LIN {X 103.987,Y -19.308,Z -79.149,A -90.000,B 90.000,C 0.000} C_DIS
LIN {X 103.058,Y -19.308,Z -80.726,A -90.000,B 90.000,C 0.000} C_DIS
LIN {X 102.198,Y -19.308,Z -82.078,A -90.000,B 90.000,C 0.000} C_DIS
LIN {X 99.737,Y -19.308,Z -85.762,A -90.000,B 90.000,C 0.000} C_DIS
LIN {X 99.864,Y -19.308,Z -87.386,A -90.000,B 90.000,C 0.000} C_DIS
LIN {X 100.040,Y -19.308,Z -89.899,A -90.000,B 90.000,C 0.000} C_DIS
LIN {X 100.045,Y -19.308,Z -89.957,A -90.000,B 90.000,C 0.000} C_DIS
LIN {X 100.412,Y -19.308,Z -91.345,A -90.000,B 90.000,C 0.000} C_DIS
LIN {X 100.428,Y -19.308,Z -91.411,A -90.000,B 90.000,C 0.000} C_DIS
LIN {X 100.504,Y -19.308,Z -91.700,A -90.000,B 90.000,C 0.000} C_DIS
LIN {X 100.648,Y -19.308,Z -92.531,A -90.000,B 90.000,C 0.000} C_DIS
LIN {X 100.763,Y -19.308,Z -93.019,A -90.000,B 90.000,C 0.000} C_DIS
LIN {X 100.838,Y -19.308,Z -93.500,A -90.000,B 90.000,C 0.000} C_DIS
LIN {X 100.877,Y -19.308,Z -93.994,A -90.000,B 90.000,C 0.000} C_DIS
LIN {X 100.998,Y -19.308,Z -94.813,A -90.000,B 90.000,C 0.000} C_DIS
LIN {X 101.014,Y -19.308,Z -95.123,A -90.000,B 90.000,C 0.000} C_DIS
LIN {X 101.095,Y -19.308,Z -96.027,A -90.000,B 90.000,C 0.000} C_DIS
LIN {X 101.110,Y -19.308,Z -96.320,A -90.000,B 90.000,C 0.000} C_DIS
LIN {X 101.175,Y -19.308,Z -97.267,A -90.000,B 90.000,C 0.000} C_DIS
LIN {X 101.202,Y -19.308,Z -97.483,A -90.000,B 90.000,C 0.000} C_DIS
LIN {X 101.290,Y -19.308,Z -98.618,A -90.000,B 90.000,C 0.000} C_DIS
LIN {X 101.319,Y -19.308,Z -98.809,A -90.000,B 90.000,C 0.000} C_DIS
LIN {X 101.430,Y -19.308,Z -100.112,A -90.000,B 90.000,C 0.000} C_DIS
LIN {X 101.445,Y -19.308,Z -100.208,A -90.000,B 90.000,C 0.000} C_DIS
LIN {X 101.588,Y -19.308,Z -101.701,A -90.000,B 90.000,C 0.000} C_DIS
LIN {X 101.643,Y -19.308,Z -102.068,A -90.000,B 90.000,C 0.000} C_DIS
LIN {X 101.782,Y -19.308,Z -103.351,A -90.000,B 90.000,C 0.000} C_DIS
LIN {X 101.920,Y -19.308,Z -104.378,A -90.000,B 90.000,C 0.000} C_DIS
LIN {X 102.259,Y -19.308,Z -106.543,A -90.000,B 90.000,C 0.000} C_DIS
LIN {X 102.427,Y -19.308,Z -107.635,A -90.000,B 90.000,C 0.000} C_DIS
LIN {X 102.586,Y -19.308,Z -108.751,A -90.000,B 90.000,C 0.000} C_DIS
LIN {X 102.776,Y -19.308,Z -110.166,A -90.000,B 90.000,C 0.000} C_DIS
LIN {X 103.011,Y -19.308,Z -111.971,A -90.000,B 90.000,C 0.000} C_DIS
LIN {X 103.313,Y -19.308,Z -114.380,A -90.000,B 90.000,C 0.000} C_DIS
LIN {X 103.602,Y -19.308,Z -116.737,A -90.000,B 90.000,C 0.000} C_DIS
LIN {X 103.814,Y -19.308,Z -118.582,A -90.000,B 90.000,C 0.000} C_DIS
LIN {X 103.886,Y -19.308,Z -119.181,A -90.000,B 90.000,C 0.000} C_DIS
LIN {X 104.063,Y -19.308,Z -120.883,A -90.000,B 90.000,C 0.000} C_DIS
LIN {X 104.148,Y -19.308,Z -121.663,A -90.000,B 90.000,C 0.000} C_DIS
LIN {X 104.284,Y -19.308,Z -123.195,A -90.000,B 90.000,C 0.000} C_DIS
LIN {X 104.370,Y -19.308,Z -124.134,A -90.000,B 90.000,C 0.000} C_DIS
LIN {X 104.532,Y -19.308,Z -126.543,A -90.000,B 90.000,C 0.000} C_DIS
LIN {X 104.557,Y -19.308,Z -127.010,A -90.000,B 90.000,C 0.000} C_DIS
LIN {X 104.601,Y -19.308,Z -128.190,A -90.000,B 90.000,C 0.000} C_DIS
LIN {X 104.655,Y -19.308,Z -129.468,A -90.000,B 90.000,C 0.000} C_DIS
LIN {X 104.668,Y -19.308,Z -130.834,A -90.000,B 90.000,C 0.000} C_DIS
LIN {X 104.688,Y -19.308,Z -132.086,A -90.000,B 90.000,C 0.000} C_DIS
LIN {X 104.665,Y -19.308,Z -133.696,A -90.000,B 90.000,C 0.000} C_DIS
LIN {X 104.655,Y -19.308,Z -134.974,A -90.000,B 90.000,C 0.000} C_DIS
LIN {X 104.619,Y -19.308,Z -136.319,A -90.000,B 90.000,C 0.000} C_DIS
LIN {X 104.547,Y -19.308,Z -138.447,A -90.000,B 90.000,C 0.000} C_DIS
LIN {X 104.485,Y -19.308,Z -139.937,A -90.000,B 90.000,C 0.000} C_DIS
LIN {X 104.383,Y -19.308,Z -142.127,A -90.000,B 90.000,C 0.000} C_DIS
LIN {X 104.310,Y -19.308,Z -143.499,A -90.000,B 90.000,C 0.000} C_DIS
LIN {X 104.174,Y -19.308,Z -145.853,A -90.000,B 90.000,C 0.000} C_DIS
LIN {X 104.083,Y -19.308,Z -147.291,A -90.000,B 90.000,C 0.000} C_DIS
LIN {X 103.924,Y -19.308,Z -149.658,A -90.000,B 90.000,C 0.000} C_DIS
LIN {X 103.809,Y -19.308,Z -151.181,A -90.000,B 90.000,C 0.000} C_DIS
LIN {X 103.665,Y -19.308,Z -153.152,A -90.000,B 90.000,C 0.000} C_DIS
LIN {X 103.314,Y -19.308,Z -157.499,A -90.000,B 90.000,C 0.000} C_DIS
LIN {X 102.978,Y -19.308,Z -161.384,A -90.000,B 90.000,C 0.000} C_DIS
LIN {X 102.664,Y -19.308,Z -164.871,A -90.000,B 90.000,C 0.000} C_DIS
LIN {X 102.336,Y -19.308,Z -168.404,A -90.000,B 90.000,C 0.000} C_DIS
LIN {X 102.004,Y -19.308,Z -171.823,A -90.000,B 90.000,C 0.000} C_DIS
LIN {X 101.666,Y -19.308,Z -175.075,A -90.000,B 90.000,C 0.000} C_DIS
LIN {X 101.590,Y -19.308,Z -175.741,A -90.000,B 90.000,C 0.000} C_DIS
LIN {X 101.303,Y -19.308,Z -178.170,A -90.000,B 90.000,C 0.000} C_DIS
LIN {X 100.894,Y -19.308,Z -181.246,A -90.000,B 90.000,C 0.000} C_DIS
LIN {X 100.474,Y -19.308,Z -184.127,A -90.000,B 90.000,C 0.000} C_DIS
LIN {X 100.075,Y -19.308,Z -186.713,A -90.000,B 90.000,C 0.000} C_DIS
LIN {X 99.715,Y -19.308,Z -189.013,A -90.000,B 90.000,C 0.000} C_DIS
LIN {X 99.354,Y -19.308,Z -191.397,A -90.000,B 90.000,C 0.000} C_DIS
LIN {X 99.271,Y -19.308,Z -191.933,A -90.000,B 90.000,C 0.000} C_DIS
LIN {X 98.939,Y -19.308,Z -193.967,A -90.000,B 90.000,C 0.000} C_DIS
LIN {X 98.678,Y -19.308,Z -195.458,A -90.000,B 90.000,C 0.000} C_DIS
LIN {X 98.423,Y -19.308,Z -196.834,A -90.000,B 90.000,C 0.000} C_DIS
LIN {X 98.011,Y -19.308,Z -198.956,A -90.000,B 90.000,C 0.000} C_DIS
LIN {X 97.713,Y -19.308,Z -200.366,A -90.000,B 90.000,C 0.000} C_DIS
LIN {X 97.101,Y -19.308,Z -203.218,A -90.000,B 90.000,C 0.000} C_DIS
LIN {X 96.760,Y -19.308,Z -204.668,A -90.000,B 90.000,C 0.000} C_DIS
LIN {X 95.957,Y -19.308,Z -208.195,A -90.000,B 90.000,C 0.000} C_DIS
LIN {X 95.642,Y -19.308,Z -209.516,A -90.000,B 90.000,C 0.000} C_DIS
LIN {X 95.578,Y -19.308,Z -209.775,A -90.000,B 90.000,C 0.000} C_DIS
LIN {X 94.321,Y -19.308,Z -215.060,A -90.000,B 90.000,C 0.000} C_DIS
LIN {X 92.959,Y -19.308,Z -220.548,A -90.000,B 90.000,C 0.000} C_DIS
LIN {X 91.672,Y -19.308,Z -225.536,A -90.000,B 90.000,C 0.000} C_DIS
LIN {X 91.541,Y -19.308,Z -226.056,A -90.000,B 90.000,C 0.000} C_DIS
LIN {X 89.987,Y -19.308,Z -231.676,A -90.000,B 90.000,C 0.000} C_DIS
LIN {X 88.154,Y -19.308,Z -237.735,A -90.000,B 90.000,C 0.000} C_DIS
LIN {X 88.090,Y -19.308,Z -237.937,A -90.000,B 90.000,C 0.000} C_DIS
LIN {X 86.454,Y -19.308,Z -242.832,A -90.000,B 90.000,C 0.000} C_DIS
LIN {X 86.214,Y -19.308,Z -243.561,A -90.000,B 90.000,C 0.000} C_DIS
LIN {X 86.214,Y -60.000,Z -243.561,A -90.000,B 90.000,C 0.000} C_DIS
LIN {X 100.091,Y -60.000,Z -90.101,A -90.000,B 90.000,C 0.000} C_DIS
LIN {X 100.091,Y -17.308,Z -90.101,A -90.000,B 90.000,C 0.000} C_DIS
LIN {X 100.230,Y -17.309,Z -90.520,A -90.000,B 90.000,C 0.000} C_DIS
LIN {X 100.336,Y -17.309,Z -90.804,A -90.000,B 90.000,C 0.000} C_DIS
LIN {X 100.668,Y -17.314,Z -91.753,A -90.000,B 90.000,C 0.000} C_DIS
LIN {X 100.794,Y -17.318,Z -92.235,A -90.000,B 90.000,C 0.000} C_DIS
LIN {X 100.884,Y -17.319,Z -92.622,A -90.000,B 90.000,C 0.000} C_DIS
LIN {X 100.988,Y -17.321,Z -92.984,A -90.000,B 90.000,C 0.000} C_DIS
LIN {X 101.100,Y -17.327,Z -93.411,A -90.000,B 90.000,C 0.000} C_DIS
LIN {X 101.168,Y -17.331,Z -93.853,A -90.000,B 90.000,C 0.000} C_DIS
LIN {X 101.322,Y -17.339,Z -94.610,A -90.000,B 90.000,C 0.000} C_DIS
LIN {X 101.351,Y -17.340,Z -94.795,A -90.000,B 90.000,C 0.000} C_DIS
LIN {X 101.396,Y -17.345,Z -95.095,A -90.000,B 90.000,C 0.000} C_DIS
LIN {X 101.414,Y -17.345,Z -95.293,A -90.000,B 90.000,C 0.000} C_DIS
LIN {X 101.528,Y -17.355,Z -96.069,A -90.000,B 90.000,C 0.000} C_DIS
LIN {X 101.546,Y -17.358,Z -96.196,A -90.000,B 90.000,C 0.000} C_DIS
LIN {X 101.560,Y -17.358,Z -96.404,A -90.000,B 90.000,C 0.000} C_DIS
LIN {X 101.676,Y -17.369,Z -97.317,A -90.000,B 90.000,C 0.000} C_DIS
LIN {X 101.756,Y -17.377,Z -97.898,A -90.000,B 90.000,C 0.000} C_DIS
LIN {X 101.825,Y -17.386,Z -98.396,A -90.000,B 90.000,C 0.000} C_DIS
LIN {X 101.854,Y -17.387,Z -98.629,A -90.000,B 90.000,C 0.000} C_DIS
LIN {X 101.860,Y -17.387,Z -98.688,A -90.000,B 90.000,C 0.000} C_DIS
LIN {X 101.918,Y -17.392,Z -99.080,A -90.000,B 90.000,C 0.000} C_DIS
LIN {X 102.046,Y -17.409,Z -99.960,A -90.000,B 90.000,C 0.000} C_DIS
LIN {X 102.058,Y -17.408,Z -100.094,A -90.000,B 90.000,C 0.000} C_DIS
LIN {X 102.260,Y -17.433,Z -101.436,A -90.000,B 90.000,C 0.000} C_DIS
LIN {X 102.287,Y -17.431,Z -101.711,A -90.000,B 90.000,C 0.000} C_DIS
LIN {X 102.331,Y -17.432,Z -101.994,A -90.000,B 90.000,C 0.000} C_DIS
LIN {X 102.532,Y -17.453,Z -103.332,A -90.000,B 90.000,C 0.000} C_DIS
LIN {X 102.578,Y -17.454,Z -103.640,A -90.000,B 90.000,C 0.000} C_DIS
LIN {X 102.603,Y -17.453,Z -103.849,A -90.000,B 90.000,C 0.000} C_DIS
LIN {X 102.667,Y -17.457,Z -104.269,A -90.000,B 90.000,C 0.000} C_DIS
LIN {X 102.901,Y -17.457,Z -105.750,A -90.000,B 90.000,C 0.000} C_DIS
LIN {X 103.122,Y -17.455,Z -107.208,A -90.000,B 90.000,C 0.000} C_DIS
LIN {X 103.352,Y -17.458,Z -108.760,A -90.000,B 90.000,C 0.000} C_DIS
LIN {X 103.439,Y -17.459,Z -109.387,A -90.000,B 90.000,C 0.000} C_DIS
LIN {X 103.665,Y -17.461,Z -111.052,A -90.000,B 90.000,C 0.000} C_DIS
LIN {X 103.740,Y -17.462,Z -111.617,A -90.000,B 90.000,C 0.000} C_DIS
LIN {X 104.045,Y -17.461,Z -114.051,A -90.000,B 90.000,C 0.000} C_DIS
LIN {X 104.152,Y -17.457,Z -115.015,A -90.000,B 90.000,C 0.000} C_DIS
LIN {X 104.226,Y -17.455,Z -115.644,A -90.000,B 90.000,C 0.000} C_DIS
LIN {X 104.332,Y -17.453,Z -116.545,A -90.000,B 90.000,C 0.000} C_DIS
LIN {X 104.387,Y -17.450,Z -117.097,A -90.000,B 90.000,C 0.000} C_DIS
LIN {X 104.604,Y -17.443,Z -119.102,A -90.000,B 90.000,C 0.000} C_DIS
LIN {X 104.811,Y -17.437,Z -121.240,A -90.000,B 90.000,C 0.000} C_DIS
LIN {X 104.850,Y -17.436,Z -121.606,A -90.000,B 90.000,C 0.000} C_DIS
LIN {X 105.001,Y -17.432,Z -123.421,A -90.000,B 90.000,C 0.000} C_DIS
LIN {X 105.063,Y -17.432,Z -124.100,A -90.000,B 90.000,C 0.000} C_DIS
LIN {X 105.228,Y -17.433,Z -126.534,A -90.000,B 90.000,C 0.000} C_DIS
LIN {X 105.256,Y -17.433,Z -127.072,A -90.000,B 90.000,C 0.000} C_DIS
LIN {X 105.363,Y -17.438,Z -129.492,A -90.000,B 90.000,C 0.000} C_DIS
LIN {X 105.387,Y -17.442,Z -130.825,A -90.000,B 90.000,C 0.000} C_DIS
LIN {X 105.414,Y -17.445,Z -132.132,A -90.000,B 90.000,C 0.000} C_DIS
LIN {X 105.404,Y -17.450,Z -133.704,A -90.000,B 90.000,C 0.000} C_DIS
LIN {X 105.400,Y -17.453,Z -135.091,A -90.000,B 90.000,C 0.000} C_DIS
LIN {X 105.360,Y -17.458,Z -136.853,A -90.000,B 90.000,C 0.000} C_DIS
LIN {X 105.316,Y -17.462,Z -138.473,A -90.000,B 90.000,C 0.000} C_DIS
LIN {X 105.222,Y -17.468,Z -140.956,A -90.000,B 90.000,C 0.000} C_DIS
LIN {X 105.169,Y -17.472,Z -142.260,A -90.000,B 90.000,C 0.000} C_DIS
LIN {X 105.092,Y -17.474,Z -143.764,A -90.000,B 90.000,C 0.000} C_DIS
LIN {X 104.980,Y -17.478,Z -145.900,A -90.000,B 90.000,C 0.000} C_DIS
LIN {X 104.775,Y -17.481,Z -149.127,A -90.000,B 90.000,C 0.000} C_DIS
LIN {X 104.729,Y -17.482,Z -149.845,A -90.000,B 90.000,C 0.000} C_DIS
LIN {X 104.440,Y -17.481,Z -153.671,A -90.000,B 90.000,C 0.000} C_DIS
LIN {X 104.110,Y -17.475,Z -157.564,A -90.000,B 90.000,C 0.000} C_DIS
LIN {X 103.752,Y -17.466,Z -161.459,A -90.000,B 90.000,C 0.000} C_DIS
LIN {X 103.351,Y -17.454,Z -165.582,A -90.000,B 90.000,C 0.000} C_DIS
LIN {X 102.981,Y -17.446,Z -169.296,A -90.000,B 90.000,C 0.000} C_DIS
LIN {X 102.710,Y -17.440,Z -171.918,A -90.000,B 90.000,C 0.000} C_DIS
LIN {X 102.535,Y -17.436,Z -173.522,A -90.000,B 90.000,C 0.000} C_DIS
LIN {X 102.352,Y -17.432,Z -175.180,A -90.000,B 90.000,C 0.000} C_DIS
LIN {X 101.981,Y -17.429,Z -178.250,A -90.000,B 90.000,C 0.000} C_DIS
LIN {X 101.603,Y -17.426,Z -181.040,A -90.000,B 90.000,C 0.000} C_DIS
LIN {X 101.539,Y -17.425,Z -181.488,A -90.000,B 90.000,C 0.000} C_DIS
LIN {X 101.155,Y -17.423,Z -184.085,A -90.000,B 90.000,C 0.000} C_DIS
LIN {X 100.474,Y -17.418,Z -188.393,A -90.000,B 90.000,C 0.000} C_DIS
LIN {X 100.361,Y -17.418,Z -189.114,A -90.000,B 90.000,C 0.000} C_DIS
LIN {X 99.996,Y -17.417,Z -191.494,A -90.000,B 90.000,C 0.000} C_DIS
LIN {X 99.965,Y -17.416,Z -191.688,A -90.000,B 90.000,C 0.000} C_DIS
LIN {X 99.583,Y -17.418,Z -194.072,A -90.000,B 90.000,C 0.000} C_DIS
LIN {X 99.476,Y -17.419,Z -194.709,A -90.000,B 90.000,C 0.000} C_DIS
LIN {X 99.324,Y -17.419,Z -195.572,A -90.000,B 90.000,C 0.000} C_DIS
LIN {X 99.078,Y -17.423,Z -196.955,A -90.000,B 90.000,C 0.000} C_DIS
LIN {X 98.888,Y -17.427,Z -198.002,A -90.000,B 90.000,C 0.000} C_DIS
LIN {X 98.676,Y -17.427,Z -199.085,A -90.000,B 90.000,C 0.000} C_DIS
LIN {X 98.394,Y -17.433,Z -200.509,A -90.000,B 90.000,C 0.000} C_DIS
LIN {X 98.106,Y -17.443,Z -201.970,A -90.000,B 90.000,C 0.000} C_DIS
LIN {X 97.805,Y -17.442,Z -203.369,A -90.000,B 90.000,C 0.000} C_DIS
LIN {X 97.484,Y -17.452,Z -204.839,A -90.000,B 90.000,C 0.000} C_DIS
LIN {X 97.050,Y -17.466,Z -206.904,A -90.000,B 90.000,C 0.000} C_DIS
LIN {X 96.867,Y -17.471,Z -207.754,A -90.000,B 90.000,C 0.000} C_DIS
LIN {X 96.726,Y -17.470,Z -208.370,A -90.000,B 90.000,C 0.000} C_DIS
LIN {X 96.421,Y -17.475,Z -209.701,A -90.000,B 90.000,C 0.000} C_DIS
LIN {X 95.655,Y -17.498,Z -213.123,A -90.000,B 90.000,C 0.000} C_DIS
LIN {X 95.147,Y -17.498,Z -215.256,A -90.000,B 90.000,C 0.000} C_DIS
LIN {X 94.309,Y -17.515,Z -218.783,A -90.000,B 90.000,C 0.000} C_DIS
LIN {X 93.950,Y -17.518,Z -220.254,A -90.000,B 90.000,C 0.000} C_DIS
LIN {X 93.823,Y -17.517,Z -220.763,A -90.000,B 90.000,C 0.000} C_DIS
LIN {X 93.724,Y -17.517,Z -221.147,A -90.000,B 90.000,C 0.000} C_DIS
LIN {X 92.458,Y -17.526,Z -226.130,A -90.000,B 90.000,C 0.000} C_DIS
LIN {X 92.352,Y -17.525,Z -226.517,A -90.000,B 90.000,C 0.000} C_DIS
LIN {X 90.897,Y -17.526,Z -231.788,A -90.000,B 90.000,C 0.000} C_DIS
LIN {X 90.724,Y -17.524,Z -232.363,A -90.000,B 90.000,C 0.000} C_DIS
LIN {X 89.062,Y -17.525,Z -237.861,A -90.000,B 90.000,C 0.000} C_DIS
LIN {X 88.983,Y -17.524,Z -238.109,A -90.000,B 90.000,C 0.000} C_DIS
LIN {X 87.179,Y -17.531,Z -243.561,A -90.000,B 90.000,C 0.000} C_DIS
LIN {X 87.179,Y -60.000,Z -243.561,A -90.000,B 90.000,C 0.000} C_DIS
LIN {X -110.313,Y -60.000,Z -243.561,A -90.000,B 90.000,C 0.000} C_DIS
LIN {X -110.313,Y -18.479,Z -243.561,A -90.000,B 90.000,C 0.000} C_DIS
LIN {X -110.301,Y -18.455,Z -243.517,A -90.000,B 90.000,C 0.000} C_DIS
LIN {X -110.261,Y -18.391,Z -243.388,A -90.000,B 90.000,C 0.000} C_DIS
LIN {X -110.203,Y -18.323,Z -243.242,A -90.000,B 90.000,C 0.000} C_DIS
LIN {X -110.174,Y -18.295,Z -243.177,A -90.000,B 90.000,C 0.000} C_DIS
LIN {X -109.840,Y -18.124,Z -242.677,A -90.000,B 90.000,C 0.000} C_DIS
LIN {X -109.452,Y -18.069,Z -242.319,A -90.000,B 90.000,C 0.000} C_DIS
LIN {X -109.374,Y -18.068,Z -242.263,A -90.000,B 90.000,C 0.000} C_DIS
LIN {X -108.603,Y -18.076,Z -241.732,A -90.000,B 90.000,C 0.000} C_DIS
LIN {X -106.834,Y -18.082,Z -240.498,A -90.000,B 90.000,C 0.000} C_DIS
LIN {X -100.205,Y -18.099,Z -235.847,A -90.000,B 90.000,C 0.000} C_DIS
LIN {X -97.781,Y -18.102,Z -234.146,A -90.000,B 90.000,C 0.000} C_DIS
LIN {X -93.938,Y -18.110,Z -231.476,A -90.000,B 90.000,C 0.000} C_DIS
LIN {X -89.899,Y -18.111,Z -228.673,A -90.000,B 90.000,C 0.000} C_DIS
LIN {X -89.665,Y -18.110,Z -228.511,A -90.000,B 90.000,C 0.000} C_DIS
LIN {X -87.245,Y -18.114,Z -226.866,A -90.000,B 90.000,C 0.000} C_DIS
LIN {X -81.874,Y -18.116,Z -223.210,A -90.000,B 90.000,C 0.000} C_DIS
LIN {X -81.580,Y -18.114,Z -223.011,A -90.000,B 90.000,C 0.000} C_DIS
LIN {X -76.713,Y -18.118,Z -219.783,A -90.000,B 90.000,C 0.000} C_DIS
LIN {X -73.418,Y -18.109,Z -217.608,A -90.000,B 90.000,C 0.000} C_DIS
LIN {X -70.830,Y -18.099,Z -215.910,A -90.000,B 90.000,C 0.000} C_DIS
LIN {X -65.406,Y -18.087,Z -212.367,A -90.000,B 90.000,C 0.000} C_DIS
LIN {X -60.511,Y -18.066,Z -209.130,A -90.000,B 90.000,C 0.000} C_DIS
LIN {X -58.236,Y -18.060,Z -207.634,A -90.000,B 90.000,C 0.000} C_DIS
LIN {X -57.950,Y -18.062,Z -207.444,A -90.000,B 90.000,C 0.000} C_DIS
LIN {X -51.703,Y -18.026,Z -203.201,A -90.000,B 90.000,C 0.000} C_DIS
LIN {X -51.585,Y -18.027,Z -203.119,A -90.000,B 90.000,C 0.000} C_DIS
LIN {X -46.435,Y -18.015,Z -199.479,A -90.000,B 90.000,C 0.000} C_DIS
LIN {X -46.154,Y -18.018,Z -199.276,A -90.000,B 90.000,C 0.000} C_DIS
LIN {X -43.931,Y -18.008,Z -197.626,A -90.000,B 90.000,C 0.000} C_DIS
LIN {X -41.923,Y -17.985,Z -196.152,A -90.000,B 90.000,C 0.000} C_DIS
LIN {X -41.724,Y -17.985,Z -196.003,A -90.000,B 90.000,C 0.000} C_DIS
LIN {X -40.829,Y -17.980,Z -195.324,A -90.000,B 90.000,C 0.000} C_DIS
LIN {X -38.690,Y -17.954,Z -193.683,A -90.000,B 90.000,C 0.000} C_DIS
LIN {X -38.089,Y -17.943,Z -193.227,A -90.000,B 90.000,C 0.000} C_DIS
LIN {X -36.620,Y -17.931,Z -192.090,A -90.000,B 90.000,C 0.000} C_DIS
LIN {X -34.749,Y -17.901,Z -190.626,A -90.000,B 90.000,C 0.000} C_DIS
LIN {X -32.943,Y -17.881,Z -189.202,A -90.000,B 90.000,C 0.000} C_DIS
LIN {X -31.630,Y -17.878,Z -188.178,A -90.000,B 90.000,C 0.000} C_DIS
LIN {X -31.435,Y -17.879,Z -188.023,A -90.000,B 90.000,C 0.000} C_DIS
LIN {X -30.006,Y -17.868,Z -186.865,A -90.000,B 90.000,C 0.000} C_DIS
LIN {X -28.713,Y -17.868,Z -185.829,A -90.000,B 90.000,C 0.000} C_DIS
LIN {X -28.525,Y -17.871,Z -185.673,A -90.000,B 90.000,C 0.000} C_DIS
LIN {X -27.122,Y -17.861,Z -184.479,A -90.000,B 90.000,C 0.000} C_DIS
LIN {X -25.979,Y -17.862,Z -183.517,A -90.000,B 90.000,C 0.000} C_DIS
LIN {X -24.802,Y -17.852,Z -182.443,A -90.000,B 90.000,C 0.000} C_DIS
LIN {X -23.613,Y -17.853,Z -181.372,A -90.000,B 90.000,C 0.000} C_DIS
LIN {X -23.524,Y -17.855,Z -181.286,A -90.000,B 90.000,C 0.000} C_DIS
LIN {X -22.591,Y -17.854,Z -180.371,A -90.000,B 90.000,C 0.000} C_DIS
LIN {X -21.251,Y -17.839,Z -179.039,A -90.000,B 90.000,C 0.000} C_DIS
LIN {X -21.040,Y -17.844,Z -178.818,A -90.000,B 90.000,C 0.000} C_DIS
LIN {X -20.425,Y -17.843,Z -178.154,A -90.000,B 90.000,C 0.000} C_DIS
LIN {X -19.010,Y -17.825,Z -176.606,A -90.000,B 90.000,C 0.000} C_DIS
LIN {X -18.887,Y -17.828,Z -176.463,A -90.000,B 90.000,C 0.000} C_DIS
LIN {X -18.374,Y -17.828,Z -175.846,A -90.000,B 90.000,C 0.000} C_DIS
LIN {X -17.081,Y -17.809,Z -174.270,A -90.000,B 90.000,C 0.000} C_DIS
LIN {X -16.818,Y -17.817,Z -173.925,A -90.000,B 90.000,C 0.000} C_DIS
LIN {X -16.274,Y -17.819,Z -173.186,A -90.000,B 90.000,C 0.000} C_DIS
LIN {X -15.242,Y -17.798,Z -171.754,A -90.000,B 90.000,C 0.000} C_DIS
LIN {X -15.058,Y -17.806,Z -171.475,A -90.000,B 90.000,C 0.000} C_DIS
LIN {X -14.670,Y -17.808,Z -170.864,A -90.000,B 90.000,C 0.000} C_DIS
LIN {X -13.644,Y -17.777,Z -169.200,A -90.000,B 90.000,C 0.000} C_DIS
LIN {X -13.389,Y -17.791,Z -168.737,A -90.000,B 90.000,C 0.000} C_DIS
LIN {X -13.310,Y -17.791,Z -168.587,A -90.000,B 90.000,C 0.000} C_DIS
LIN {X -12.460,Y -17.750,Z -166.906,A -90.000,B 90.000,C 0.000} C_DIS
LIN {X -12.399,Y -17.751,Z -166.777,A -90.000,B 90.000,C 0.000} C_DIS
LIN {X -12.219,Y -17.765,Z -166.355,A -90.000,B 90.000,C 0.000} C_DIS
LIN {X -11.645,Y -17.726,Z -164.814,A -90.000,B 90.000,C 0.000} C_DIS
LIN {X -11.564,Y -17.727,Z -164.573,A -90.000,B 90.000,C 0.000} C_DIS
LIN {X -11.483,Y -17.743,Z -164.266,A -90.000,B 90.000,C 0.000} C_DIS
LIN {X -11.234,Y -17.711,Z -163.012,A -90.000,B 90.000,C 0.000} C_DIS
LIN {X -11.233,Y -17.735,Z -162.809,A -90.000,B 90.000,C 0.000} C_DIS
LIN {X -11.258,Y -17.724,Z -162.439,A -90.000,B 90.000,C 0.000} C_DIS
LIN {X -11.277,Y -17.714,Z -162.137,A -90.000,B 90.000,C 0.000} C_DIS
LIN {X -11.311,Y -17.679,Z -161.927,A -90.000,B 90.000,C 0.000} C_DIS
LIN {X -11.431,Y -17.667,Z -161.591,A -90.000,B 90.000,C 0.000} C_DIS
LIN {X -11.573,Y -17.618,Z -161.265,A -90.000,B 90.000,C 0.000} C_DIS
LIN {X -11.777,Y -17.616,Z -160.935,A -90.000,B 90.000,C 0.000} C_DIS
LIN {X -12.055,Y -17.570,Z -160.529,A -90.000,B 90.000,C 0.000} C_DIS
LIN {X -12.189,Y -17.564,Z -160.370,A -90.000,B 90.000,C 0.000} C_DIS
LIN {X -12.579,Y -17.562,Z -159.895,A -90.000,B 90.000,C 0.000} C_DIS
LIN {X -12.689,Y -17.558,Z -159.753,A -90.000,B 90.000,C 0.000} C_DIS
LIN {X -12.856,Y -17.547,Z -159.541,A -90.000,B 90.000,C 0.000} C_DIS
LIN {X -12.904,Y -17.543,Z -159.475,A -90.000,B 90.000,C 0.000} C_DIS
LIN {X -13.256,Y -17.539,Z -159.079,A -90.000,B 90.000,C 0.000} C_DIS
LIN {X -13.618,Y -17.525,Z -158.677,A -90.000,B 90.000,C 0.000} C_DIS
LIN {X -13.890,Y -17.505,Z -158.340,A -90.000,B 90.000,C 0.000} C_DIS
LIN {X -14.445,Y -17.501,Z -157.763,A -90.000,B 90.000,C 0.000} C_DIS
LIN {X -14.736,Y -17.492,Z -157.465,A -90.000,B 90.000,C 0.000} C_DIS
LIN {X -15.053,Y -17.472,Z -157.099,A -90.000,B 90.000,C 0.000} C_DIS
LIN {X -15.852,Y -17.469,Z -156.326,A -90.000,B 90.000,C 0.000} C_DIS
LIN {X -16.143,Y -17.462,Z -156.031,A -90.000,B 90.000,C 0.000} C_DIS
LIN {X -16.300,Y -17.456,Z -155.872,A -90.000,B 90.000,C 0.000} C_DIS
LIN {X -16.598,Y -17.443,Z -155.560,A -90.000,B 90.000,C 0.000} C_DIS
LIN {X -17.901,Y -17.442,Z -154.370,A -90.000,B 90.000,C 0.000} C_DIS
LIN {X -18.334,Y -17.434,Z -153.951,A -90.000,B 90.000,C 0.000} C_DIS
LIN {X -18.608,Y -17.426,Z -153.686,A -90.000,B 90.000,C 0.000} C_DIS
LIN {X -20.437,Y -17.425,Z -152.079,A -90.000,B 90.000,C 0.000} C_DIS
LIN {X -21.457,Y -17.414,Z -151.147,A -90.000,B 90.000,C 0.000} C_DIS
LIN {X -21.590,Y -17.412,Z -151.026,A -90.000,B 90.000,C 0.000} C_DIS
LIN {X -23.480,Y -17.412,Z -149.291,A -90.000,B 90.000,C 0.000} C_DIS
LIN {X -24.708,Y -17.403,Z -148.131,A -90.000,B 90.000,C 0.000} C_DIS
LIN {X -25.063,Y -17.402,Z -147.781,A -90.000,B 90.000,C 0.000} C_DIS
LIN {X -27.238,Y -17.403,Z -145.567,A -90.000,B 90.000,C 0.000} C_DIS
LIN {X -28.146,Y -17.398,Z -144.626,A -90.000,B 90.000,C 0.000} C_DIS
LIN {X -28.313,Y -17.396,Z -144.448,A -90.000,B 90.000,C 0.000} C_DIS
LIN {X -28.459,Y -17.396,Z -144.284,A -90.000,B 90.000,C 0.000} C_DIS
LIN {X -31.251,Y -17.401,Z -140.928,A -90.000,B 90.000,C 0.000} C_DIS
LIN {X -31.512,Y -17.400,Z -140.610,A -90.000,B 90.000,C 0.000} C_DIS
LIN {X -31.755,Y -17.395,Z -140.285,A -90.000,B 90.000,C 0.000} C_DIS
LIN {X -31.800,Y -17.396,Z -140.223,A -90.000,B 90.000,C 0.000} C_DIS
LIN {X -31.998,Y -17.394,Z -139.910,A -90.000,B 90.000,C 0.000} C_DIS
LIN {X -33.208,Y -17.397,Z -138.027,A -90.000,B 90.000,C 0.000} C_DIS
LIN {X -34.363,Y -17.399,Z -136.214,A -90.000,B 90.000,C 0.000} C_DIS
LIN {X -34.522,Y -17.396,Z -135.946,A -90.000,B 90.000,C 0.000} C_DIS
LIN {X -35.291,Y -17.395,Z -134.451,A -90.000,B 90.000,C 0.000} C_DIS
LIN {X -36.136,Y -17.394,Z -132.804,A -90.000,B 90.000,C 0.000} C_DIS
LIN {X -36.693,Y -17.395,Z -131.712,A -90.000,B 90.000,C 0.000} C_DIS
LIN {X -36.805,Y -17.392,Z -131.461,A -90.000,B 90.000,C 0.000} C_DIS
LIN {X -37.879,Y -17.391,Z -128.993,A -90.000,B 90.000,C 0.000} C_DIS
LIN {X -38.306,Y -17.391,Z -128.012,A -90.000,B 90.000,C 0.000} C_DIS
LIN {X -38.458,Y -17.388,Z -127.638,A -90.000,B 90.000,C 0.000} C_DIS
LIN {X -39.565,Y -17.381,Z -124.911,A -90.000,B 90.000,C 0.000} C_DIS
LIN {X -39.737,Y -17.380,Z -124.479,A -90.000,B 90.000,C 0.000} C_DIS
LIN {X -40.078,Y -17.375,Z -123.681,A -90.000,B 90.000,C 0.000} C_DIS
LIN {X -40.355,Y -17.368,Z -123.027,A -90.000,B 90.000,C 0.000} C_DIS
LIN {X -40.551,Y -17.362,Z -122.565,A -90.000,B 90.000,C 0.000} C_DIS
LIN {X -40.915,Y -17.357,Z -121.814,A -90.000,B 90.000,C 0.000} C_DIS
LIN {X -41.064,Y -17.353,Z -121.508,A -90.000,B 90.000,C 0.000} C_DIS
LIN {X -41.384,Y -17.349,Z -120.906,A -90.000,B 90.000,C 0.000} C_DIS
LIN {X -41.550,Y -17.349,Z -120.630,A -90.000,B 90.000,C 0.000} C_DIS
LIN {X -41.646,Y -17.347,Z -120.472,A -90.000,B 90.000,C 0.000} C_DIS
LIN {X -42.217,Y -17.344,Z -119.585,A -90.000,B 90.000,C 0.000} C_DIS
LIN {X -42.411,Y -17.347,Z -119.318,A -90.000,B 90.000,C 0.000} C_DIS
LIN {X -42.625,Y -17.346,Z -119.027,A -90.000,B 90.000,C 0.000} C_DIS
LIN {X -43.316,Y -17.345,Z -118.108,A -90.000,B 90.000,C 0.000} C_DIS
LIN {X -44.066,Y -17.351,Z -117.176,A -90.000,B 90.000,C 0.000} C_DIS
LIN {X -45.345,Y -17.355,Z -115.589,A -90.000,B 90.000,C 0.000} C_DIS
LIN {X -47.502,Y -17.366,Z -112.941,A -90.000,B 90.000,C 0.000} C_DIS
LIN {X -48.901,Y -17.369,Z -111.186,A -90.000,B 90.000,C 0.000} C_DIS
LIN {X -50.009,Y -17.374,Z -109.806,A -90.000,B 90.000,C 0.000} C_DIS
LIN {X -50.851,Y -17.373,Z -108.717,A -90.000,B 90.000,C 0.000} C_DIS
LIN {X -51.895,Y -17.377,Z -107.362,A -90.000,B 90.000,C 0.000} C_DIS
LIN {X -52.606,Y -17.378,Z -106.436,A -90.000,B 90.000,C 0.000} C_DIS
LIN {X -52.812,Y -17.377,Z -106.158,A -90.000,B 90.000,C 0.000} C_DIS
LIN {X -53.083,Y -17.374,Z -105.789,A -90.000,B 90.000,C 0.000} C_DIS
LIN {X -54.105,Y -17.373,Z -104.390,A -90.000,B 90.000,C 0.000} C_DIS
LIN {X -54.659,Y -17.370,Z -103.630,A -90.000,B 90.000,C 0.000} C_DIS
LIN {X -55.391,Y -17.368,Z -102.640,A -90.000,B 90.000,C 0.000} C_DIS
LIN {X -55.998,Y -17.365,Z -101.794,A -90.000,B 90.000,C 0.000} C_DIS
LIN {X -57.058,Y -17.364,Z -100.341,A -90.000,B 90.000,C 0.000} C_DIS
LIN {X -57.561,Y -17.361,Z -99.651,A -90.000,B 90.000,C 0.000} C_DIS
LIN {X -58.119,Y -17.359,Z -98.896,A -90.000,B 90.000,C 0.000} C_DIS
LIN {X -58.965,Y -17.355,Z -97.746,A -90.000,B 90.000,C 0.000} C_DIS
LIN {X -59.895,Y -17.355,Z -96.509,A -90.000,B 90.000,C 0.000} C_DIS
LIN {X -60.318,Y -17.356,Z -95.953,A -90.000,B 90.000,C 0.000} C_DIS
LIN {X -61.327,Y -17.356,Z -94.642,A -90.000,B 90.000,C 0.000} C_DIS
LIN {X -61.836,Y -17.354,Z -93.978,A -90.000,B 90.000,C 0.000} C_DIS
LIN {X -62.043,Y -17.354,Z -93.713,A -90.000,B 90.000,C 0.000} C_DIS
LIN {X -62.829,Y -17.355,Z -92.738,A -90.000,B 90.000,C 0.000} C_DIS
LIN {X -63.344,Y -17.355,Z -92.100,A -90.000,B 90.000,C 0.000} C_DIS
LIN {X -64.006,Y -17.356,Z -91.284,A -90.000,B 90.000,C 0.000} C_DIS
LIN {X -64.320,Y -17.360,Z -90.921,A -90.000,B 90.000,C 0.000} C_DIS
LIN {X -64.715,Y -17.361,Z -90.465,A -90.000,B 90.000,C 0.000} C_DIS
LIN {X -65.741,Y -17.363,Z -89.269,A -90.000,B 90.000,C 0.000} C_DIS
LIN {X -66.297,Y -17.367,Z -88.666,A -90.000,B 90.000,C 0.000} C_DIS
LIN {X -67.110,Y -17.370,Z -87.782,A -90.000,B 90.000,C 0.000} C_DIS
LIN {X -67.323,Y -17.370,Z -87.551,A -90.000,B 90.000,C 0.000} C_DIS
LIN {X -67.599,Y -17.377,Z -87.283,A -90.000,B 90.000,C 0.000} C_DIS
LIN {X -67.867,Y -17.381,Z -87.018,A -90.000,B 90.000,C 0.000} C_DIS
LIN {X -69.003,Y -17.389,Z -85.867,A -90.000,B 90.000,C 0.000} C_DIS
LIN {X -69.685,Y -17.404,Z -85.221,A -90.000,B 90.000,C 0.000} C_DIS
LIN {X -70.646,Y -17.422,Z -84.311,A -90.000,B 90.000,C 0.000} C_DIS
LIN {X -70.930,Y -17.431,Z -84.056,A -90.000,B 90.000,C 0.000} C_DIS
LIN {X -71.415,Y -17.448,Z -83.627,A -90.000,B 90.000,C 0.000} C_DIS
LIN {X -71.768,Y -17.458,Z -83.316,A -90.000,B 90.000,C 0.000} C_DIS
LIN {X -72.443,Y -17.476,Z -82.714,A -90.000,B 90.000,C 0.000} C_DIS
LIN {X -72.803,Y -17.495,Z -82.421,A -90.000,B 90.000,C 0.000} C_DIS
LIN {X -73.068,Y -17.506,Z -82.206,A -90.000,B 90.000,C 0.000} C_DIS
LIN {X -74.140,Y -17.542,Z -81.346,A -90.000,B 90.000,C 0.000} C_DIS
LIN {X -74.232,Y -17.546,Z -81.275,A -90.000,B 90.000,C 0.000} C_DIS
LIN {X -74.523,Y -17.569,Z -81.071,A -90.000,B 90.000,C 0.000} C_DIS
LIN {X -75.117,Y -17.586,Z -80.674,A -90.000,B 90.000,C 0.000} C_DIS
LIN {X -75.460,Y -17.598,Z -80.451,A -90.000,B 90.000,C 0.000} C_DIS
LIN {X -75.812,Y -17.575,Z -80.249,A -90.000,B 90.000,C 0.000} C_DIS
LIN {X -75.989,Y -17.574,Z -80.165,A -90.000,B 90.000,C 0.000} C_DIS
LIN {X -76.378,Y -17.572,Z -79.985,A -90.000,B 90.000,C 0.000} C_DIS
LIN {X -77.347,Y -17.510,Z -79.572,A -90.000,B 90.000,C 0.000} C_DIS
LIN {X -78.122,Y -17.474,Z -79.275,A -90.000,B 90.000,C 0.000} C_DIS
LIN {X -78.515,Y -17.461,Z -79.122,A -90.000,B 90.000,C 0.000} C_DIS
LIN {X -78.841,Y -17.448,Z -78.988,A -90.000,B 90.000,C 0.000} C_DIS
LIN {X -79.089,Y -17.444,Z -78.890,A -90.000,B 90.000,C 0.000} C_DIS
LIN {X -79.673,Y -17.437,Z -78.652,A -90.000,B 90.000,C 0.000} C_DIS
LIN {X -80.856,Y -17.410,Z -78.129,A -90.000,B 90.000,C 0.000} C_DIS
LIN {X -81.273,Y -17.404,Z -77.912,A -90.000,B 90.000,C 0.000} C_DIS
LIN {X -81.542,Y -17.402,Z -77.765,A -90.000,B 90.000,C 0.000} C_DIS
LIN {X -82.804,Y -17.413,Z -77.108,A -90.000,B 90.000,C 0.000} C_DIS
LIN {X -83.109,Y -17.407,Z -76.921,A -90.000,B 90.000,C 0.000} C_DIS
LIN {X -83.635,Y -17.409,Z -76.592,A -90.000,B 90.000,C 0.000} C_DIS
LIN {X -83.988,Y -17.412,Z -76.367,A -90.000,B 90.000,C 0.000} C_DIS
LIN {X -84.924,Y -17.408,Z -75.703,A -90.000,B 90.000,C 0.000} C_DIS
LIN {X -85.303,Y -17.408,Z -75.431,A -90.000,B 90.000,C 0.000} C_DIS
LIN {X -85.466,Y -17.406,Z -75.303,A -90.000,B 90.000,C 0.000} C_DIS
LIN {X -85.876,Y -17.405,Z -74.994,A -90.000,B 90.000,C 0.000} C_DIS
LIN {X -86.011,Y -17.406,Z -74.889,A -90.000,B 90.000,C 0.000} C_DIS
LIN {X -86.206,Y -17.403,Z -74.740,A -90.000,B 90.000,C 0.000} C_DIS
LIN {X -86.317,Y -17.404,Z -74.660,A -90.000,B 90.000,C 0.000} C_DIS
LIN {X -86.550,Y -17.403,Z -74.481,A -90.000,B 90.000,C 0.000} C_DIS
LIN {X -86.724,Y -17.400,Z -74.349,A -90.000,B 90.000,C 0.000} C_DIS
LIN {X -86.998,Y -17.394,Z -74.132,A -90.000,B 90.000,C 0.000} C_DIS
LIN {X -87.561,Y -17.393,Z -73.712,A -90.000,B 90.000,C 0.000} C_DIS
LIN {X -87.871,Y -17.389,Z -73.466,A -90.000,B 90.000,C 0.000} C_DIS
LIN {X -88.289,Y -17.391,Z -73.133,A -90.000,B 90.000,C 0.000} C_DIS
LIN {X -88.334,Y -17.391,Z -73.098,A -90.000,B 90.000,C 0.000} C_DIS
LIN {X -89.014,Y -17.386,Z -72.526,A -90.000,B 90.000,C 0.000} C_DIS
LIN {X -89.731,Y -17.392,Z -71.914,A -90.000,B 90.000,C 0.000} C_DIS
LIN {X -90.039,Y -17.402,Z -71.665,A -90.000,B 90.000,C 0.000} C_DIS
LIN {X -90.376,Y -17.411,Z -71.380,A -90.000,B 90.000,C 0.000} C_DIS
LIN {X -90.758,Y -17.431,Z -71.095,A -90.000,B 90.000,C 0.000} C_DIS
LIN {X -90.895,Y -17.436,Z -70.986,A -90.000,B 90.000,C 0.000} C_DIS
LIN {X -91.163,Y -17.461,Z -70.812,A -90.000,B 90.000,C 0.000} C_DIS
LIN {X -91.400,Y -17.475,Z -70.645,A -90.000,B 90.000,C 0.000} C_DIS
LIN {X -91.627,Y -17.496,Z -70.507,A -90.000,B 90.000,C 0.000} C_DIS
LIN {X -91.825,Y -17.517,Z -70.383,A -90.000,B 90.000,C 0.000} C_DIS
LIN {X -92.024,Y -17.532,Z -70.264,A -90.000,B 90.000,C 0.000} C_DIS
LIN {X -92.341,Y -17.564,Z -70.083,A -90.000,B 90.000,C 0.000} C_DIS
LIN {X -92.507,Y -17.577,Z -69.991,A -90.000,B 90.000,C 0.000} C_DIS
LIN {X -92.960,Y -17.605,Z -69.723,A -90.000,B 90.000,C 0.000} C_DIS
LIN {X -93.347,Y -17.632,Z -69.507,A -90.000,B 90.000,C 0.000} C_DIS
LIN {X -93.430,Y -17.638,Z -69.460,A -90.000,B 90.000,C 0.000} C_DIS
LIN {X -93.943,Y -17.663,Z -69.144,A -90.000,B 90.000,C 0.000} C_DIS
LIN {X -94.458,Y -17.683,Z -68.833,A -90.000,B 90.000,C 0.000} C_DIS
LIN {X -94.658,Y -17.691,Z -68.703,A -90.000,B 90.000,C 0.000} C_DIS
LIN {X -94.935,Y -17.706,Z -68.526,A -90.000,B 90.000,C 0.000} C_DIS
LIN {X -95.060,Y -17.712,Z -68.444,A -90.000,B 90.000,C 0.000} C_DIS
LIN {X -95.458,Y -17.749,Z -68.212,A -90.000,B 90.000,C 0.000} C_DIS
LIN {X -95.634,Y -17.759,Z -68.092,A -90.000,B 90.000,C 0.000} C_DIS
LIN {X -95.861,Y -17.782,Z -67.946,A -90.000,B 90.000,C 0.000} C_DIS
LIN {X -95.952,Y -17.795,Z -67.895,A -90.000,B 90.000,C 0.000} C_DIS
LIN {X -96.300,Y -17.834,Z -67.679,A -90.000,B 90.000,C 0.000} C_DIS
LIN {X -96.472,Y -17.848,Z -67.564,A -90.000,B 90.000,C 0.000} C_DIS
LIN {X -96.585,Y -17.863,Z -67.495,A -90.000,B 90.000,C 0.000} C_DIS
LIN {X -97.082,Y -17.936,Z -67.183,A -90.000,B 90.000,C 0.000} C_DIS
LIN {X -97.570,Y -17.992,Z -66.855,A -90.000,B 90.000,C 0.000} C_DIS
LIN {X -98.004,Y -18.044,Z -66.560,A -90.000,B 90.000,C 0.000} C_DIS
LIN {X -98.193,Y -18.065,Z -66.434,A -90.000,B 90.000,C 0.000} C_DIS
LIN {X -98.449,Y -18.086,Z -66.246,A -90.000,B 90.000,C 0.000} C_DIS
LIN {X -99.533,Y -18.167,Z -65.440,A -90.000,B 90.000,C 0.000} C_DIS
LIN {X -99.798,Y -18.170,Z -65.228,A -90.000,B 90.000,C 0.000} C_DIS
LIN {X -100.247,Y -18.172,Z -64.867,A -90.000,B 90.000,C 0.000} C_DIS
LIN {X -100.885,Y -18.168,Z -64.365,A -90.000,B 90.000,C 0.000} C_DIS
LIN {X -101.153,Y -18.151,Z -64.134,A -90.000,B 90.000,C 0.000} C_DIS
LIN {X -101.615,Y -18.110,Z -63.725,A -90.000,B 90.000,C 0.000} C_DIS
LIN {X -101.973,Y -18.074,Z -63.421,A -90.000,B 90.000,C 0.000} C_DIS
LIN {X -102.157,Y -18.055,Z -63.260,A -90.000,B 90.000,C 0.000} C_DIS
LIN {X -102.282,Y -18.039,Z -63.148,A -90.000,B 90.000,C 0.000} C_DIS
LIN {X -102.460,Y -18.012,Z -62.980,A -90.000,B 90.000,C 0.000} C_DIS
LIN {X -103.232,Y -17.864,Z -62.203,A -90.000,B 90.000,C 0.000} C_DIS
LIN {X -103.300,Y -17.851,Z -62.130,A -90.000,B 90.000,C 0.000} C_DIS
LIN {X -103.537,Y -17.810,Z -61.868,A -90.000,B 90.000,C 0.000} C_DIS
LIN {X -103.670,Y -17.781,Z -61.707,A -90.000,B 90.000,C 0.000} C_DIS
LIN {X -104.045,Y -17.702,Z -61.244,A -90.000,B 90.000,C 0.000} C_DIS
LIN {X -104.356,Y -17.633,Z -60.845,A -90.000,B 90.000,C 0.000} C_DIS
LIN {X -104.452,Y -17.615,Z -60.716,A -90.000,B 90.000,C 0.000} C_DIS
LIN {X -104.883,Y -17.545,Z -60.105,A -90.000,B 90.000,C 0.000} C_DIS
LIN {X -104.940,Y -17.536,Z -60.024,A -90.000,B 90.000,C 0.000} C_DIS
LIN {X -105.026,Y -17.531,Z -59.925,A -90.000,B 90.000,C 0.000} C_DIS
LIN {X -105.115,Y -17.525,Z -59.817,A -90.000,B 90.000,C 0.000} C_DIS
LIN {X -105.165,Y -17.525,Z -59.764,A -90.000,B 90.000,C 0.000} C_DIS
LIN {X -105.425,Y -17.518,Z -59.465,A -90.000,B 90.000,C 0.000} C_DIS
LIN {X -105.641,Y -17.514,Z -59.215,A -90.000,B 90.000,C 0.000} C_DIS
LIN {X -105.958,Y -17.522,Z -58.864,A -90.000,B 90.000,C 0.000} C_DIS
LIN {X -106.093,Y -17.522,Z -58.701,A -90.000,B 90.000,C 0.000} C_DIS
LIN {X -106.415,Y -17.532,Z -58.312,A -90.000,B 90.000,C 0.000} C_DIS
LIN {X -106.591,Y -17.540,Z -58.105,A -90.000,B 90.000,C 0.000} C_DIS
LIN {X -106.768,Y -17.545,Z -57.881,A -90.000,B 90.000,C 0.000} C_DIS
LIN {X -106.962,Y -17.550,Z -57.646,A -90.000,B 90.000,C 0.000} C_DIS
LIN {X -107.051,Y -17.552,Z -57.529,A -90.000,B 90.000,C 0.000} C_DIS
LIN {X -107.142,Y -17.557,Z -57.413,A -90.000,B 90.000,C 0.000} C_DIS
LIN {X -107.260,Y -17.562,Z -57.256,A -90.000,B 90.000,C 0.000} C_DIS
LIN {X -107.440,Y -17.578,Z -57.010,A -90.000,B 90.000,C 0.000} C_DIS
LIN {X -107.576,Y -17.588,Z -56.819,A -90.000,B 90.000,C 0.000} C_DIS
LIN {X -107.736,Y -17.603,Z -56.599,A -90.000,B 90.000,C 0.000} C_DIS
LIN {X -107.811,Y -17.610,Z -56.487,A -90.000,B 90.000,C 0.000} C_DIS
LIN {X -107.902,Y -17.622,Z -56.351,A -90.000,B 90.000,C 0.000} C_DIS
LIN {X -108.154,Y -17.653,Z -55.949,A -90.000,B 90.000,C 0.000} C_DIS
LIN {X -108.447,Y -17.681,Z -55.429,A -90.000,B 90.000,C 0.000} C_DIS
LIN {X -108.576,Y -17.698,Z -55.187,A -90.000,B 90.000,C 0.000} C_DIS
LIN {X -108.664,Y -17.718,Z -55.017,A -90.000,B 90.000,C 0.000} C_DIS
LIN {X -108.914,Y -17.768,Z -54.496,A -90.000,B 90.000,C 0.000} C_DIS
LIN {X -109.056,Y -17.798,Z -54.131,A -90.000,B 90.000,C 0.000} C_DIS
LIN {X -109.149,Y -17.820,Z -53.881,A -90.000,B 90.000,C 0.000} C_DIS
LIN {X -109.341,Y -17.867,Z -53.367,A -90.000,B 90.000,C 0.000} C_DIS
LIN {X -109.388,Y -17.880,Z -53.237,A -90.000,B 90.000,C 0.000} C_DIS
LIN {X -109.418,Y -17.891,Z -53.137,A -90.000,B 90.000,C 0.000} C_DIS
LIN {X -109.516,Y -17.925,Z -52.775,A -90.000,B 90.000,C 0.000} C_DIS
LIN {X -109.578,Y -17.937,Z -52.486,A -90.000,B 90.000,C 0.000} C_DIS
LIN {X -109.649,Y -17.954,Z -52.132,A -90.000,B 90.000,C 0.000} C_DIS
LIN {X -109.706,Y -17.967,Z -51.807,A -90.000,B 90.000,C 0.000} C_DIS
LIN {X -109.719,Y -17.973,Z -51.713,A -90.000,B 90.000,C 0.000} C_DIS
LIN {X -109.754,Y -17.980,Z -51.396,A -90.000,B 90.000,C 0.000} C_DIS
LIN {X -109.770,Y -17.990,Z -51.194,A -90.000,B 90.000,C 0.000} C_DIS
LIN {X -109.777,Y -17.996,Z -51.099,A -90.000,B 90.000,C 0.000} C_DIS
LIN {X -109.779,Y -17.998,Z -50.942,A -90.000,B 90.000,C 0.000} C_DIS
LIN {X -109.776,Y -18.006,Z -50.659,A -90.000,B 90.000,C 0.000} C_DIS
LIN {X -109.774,Y -18.007,Z -50.592,A -90.000,B 90.000,C 0.000} C_DIS
LIN {X -109.753,Y -17.999,Z -50.276,A -90.000,B 90.000,C 0.000} C_DIS
LIN {X -109.731,Y -17.998,Z -50.053,A -90.000,B 90.000,C 0.000} C_DIS
LIN {X -109.685,Y -18.009,Z -49.727,A -90.000,B 90.000,C 0.000} C_DIS
LIN {X -109.603,Y -17.999,Z -49.326,A -90.000,B 90.000,C 0.000} C_DIS
LIN {X -109.542,Y -17.990,Z -49.073,A -90.000,B 90.000,C 0.000} C_DIS
LIN {X -109.497,Y -17.990,Z -48.912,A -90.000,B 90.000,C 0.000} C_DIS
LIN {X -109.469,Y -17.993,Z -48.814,A -90.000,B 90.000,C 0.000} C_DIS
LIN {X -109.398,Y -17.988,Z -48.604,A -90.000,B 90.000,C 0.000} C_DIS
LIN {X -109.336,Y -17.987,Z -48.431,A -90.000,B 90.000,C 0.000} C_DIS
LIN {X -109.243,Y -17.984,Z -48.205,A -90.000,B 90.000,C 0.000} C_DIS
LIN {X -109.226,Y -17.984,Z -48.168,A -90.000,B 90.000,C 0.000} C_DIS
LIN {X -109.232,Y -17.925,Z -48.044,A -90.000,B 90.000,C 0.000} C_DIS
LIN {X -109.234,Y -17.894,Z -47.973,A -90.000,B 90.000,C 0.000} C_DIS
LIN {X -109.231,Y -17.819,Z -47.808,A -90.000,B 90.000,C 0.000} C_DIS
LIN {X -109.226,Y -17.775,Z -47.708,A -90.000,B 90.000,C 0.000} C_DIS
LIN {X -109.211,Y -17.694,Z -47.514,A -90.000,B 90.000,C 0.000} C_DIS
LIN {X -109.192,Y -17.636,Z -47.370,A -90.000,B 90.000,C 0.000} C_DIS
LIN {X -109.172,Y -17.594,Z -47.256,A -90.000,B 90.000,C 0.000} C_DIS
LIN {X -109.310,Y -17.607,Z -47.007,A -90.000,B 90.000,C 0.000} C_DIS
LIN {X -109.469,Y -17.623,Z -46.712,A -90.000,B 90.000,C 0.000} C_DIS
LIN {X -109.626,Y -17.635,Z -46.398,A -90.000,B 90.000,C 0.000} C_DIS
LIN {X -109.732,Y -17.645,Z -46.181,A -90.000,B 90.000,C 0.000} C_DIS
LIN {X -109.816,Y -17.651,Z -45.987,A -90.000,B 90.000,C 0.000} C_DIS
LIN {X -109.986,Y -17.670,Z -45.584,A -90.000,B 90.000,C 0.000} C_DIS
LIN {X -110.184,Y -17.705,Z -45.087,A -90.000,B 90.000,C 0.000} C_DIS
LIN {X -110.247,Y -17.721,Z -44.919,A -90.000,B 90.000,C 0.000} C_DIS
LIN {X -110.280,Y -17.728,Z -44.813,A -90.000,B 90.000,C 0.000} C_DIS
LIN {X -110.351,Y -17.742,Z -44.573,A -90.000,B 90.000,C 0.000} C_DIS
LIN {X -110.480,Y -17.775,Z -44.114,A -90.000,B 90.000,C 0.000} C_DIS
LIN {X -110.500,Y -17.782,Z -44.034,A -90.000,B 90.000,C 0.000} C_DIS
LIN {X -110.582,Y -17.806,Z -43.642,A -90.000,B 90.000,C 0.000} C_DIS
LIN {X -110.628,Y -17.817,Z -43.395,A -90.000,B 90.000,C 0.000} C_DIS
LIN {X -110.637,Y -17.822,Z -43.336,A -90.000,B 90.000,C 0.000} C_DIS
LIN {X -110.698,Y -17.851,Z -42.958,A -90.000,B 90.000,C 0.000} C_DIS
LIN {X -110.705,Y -17.857,Z -42.907,A -90.000,B 90.000,C 0.000} C_DIS
LIN {X -110.741,Y -17.883,Z -42.552,A -90.000,B 90.000,C 0.000} C_DIS
LIN {X -110.750,Y -17.898,Z -42.333,A -90.000,B 90.000,C 0.000} C_DIS
LIN {X -110.756,Y -17.912,Z -42.155,A -90.000,B 90.000,C 0.000} C_DIS
LIN {X -110.755,Y -17.946,Z -41.664,A -90.000,B 90.000,C 0.000} C_DIS
LIN {X -110.746,Y -17.959,Z -41.494,A -90.000,B 90.000,C 0.000} C_DIS
LIN {X -110.728,Y -17.981,Z -41.256,A -90.000,B 90.000,C 0.000} C_DIS
LIN {X -110.691,Y -18.002,Z -40.942,A -90.000,B 90.000,C 0.000} C_DIS
LIN {X -110.664,Y -18.010,Z -40.757,A -90.000,B 90.000,C 0.000} C_DIS
LIN {X -110.633,Y -18.022,Z -40.581,A -90.000,B 90.000,C 0.000} C_DIS
LIN {X -110.565,Y -18.043,Z -40.280,A -90.000,B 90.000,C 0.000} C_DIS
LIN {X -110.455,Y -18.060,Z -39.890,A -90.000,B 90.000,C 0.000} C_DIS
LIN {X -110.415,Y -18.066,Z -39.765,A -90.000,B 90.000,C 0.000} C_DIS
LIN {X -110.370,Y -18.075,Z -39.634,A -90.000,B 90.000,C 0.000} C_DIS
LIN {X -110.286,Y -18.084,Z -39.414,A -90.000,B 90.000,C 0.000} C_DIS
LIN {X -110.158,Y -18.103,Z -39.108,A -90.000,B 90.000,C 0.000} C_DIS
LIN {X -110.104,Y -18.110,Z -38.985,A -90.000,B 90.000,C 0.000} C_DIS
LIN {X -109.980,Y -18.119,Z -38.728,A -90.000,B 90.000,C 0.000} C_DIS
LIN {X -109.920,Y -18.124,Z -38.617,A -90.000,B 90.000,C 0.000} C_DIS
LIN {X -109.797,Y -18.141,Z -38.405,A -90.000,B 90.000,C 0.000} C_DIS
LIN {X -109.763,Y -18.143,Z -38.348,A -90.000,B 90.000,C 0.000} C_DIS
LIN {X -109.673,Y -18.146,Z -38.210,A -90.000,B 90.000,C 0.000} C_DIS
LIN {X -109.463,Y -18.157,Z -37.908,A -90.000,B 90.000,C 0.000} C_DIS
LIN {X -109.423,Y -18.161,Z -37.855,A -90.000,B 90.000,C 0.000} C_DIS
LIN {X -109.188,Y -18.162,Z -37.576,A -90.000,B 90.000,C 0.000} C_DIS
LIN {X -109.147,Y -18.163,Z -37.529,A -90.000,B 90.000,C 0.000} C_DIS
LIN {X -109.073,Y -18.166,Z -37.453,A -90.000,B 90.000,C 0.000} C_DIS
LIN {X -108.970,Y -18.172,Z -37.351,A -90.000,B 90.000,C 0.000} C_DIS
LIN {X -108.671,Y -18.170,Z -37.077,A -90.000,B 90.000,C 0.000} C_DIS
LIN {X -108.592,Y -18.164,Z -37.010,A -90.000,B 90.000,C 0.000} C_DIS
LIN {X -108.443,Y -18.158,Z -36.895,A -90.000,B 90.000,C 0.000} C_DIS
LIN {X -108.280,Y -18.156,Z -36.778,A -90.000,B 90.000,C 0.000} C_DIS
LIN {X -108.133,Y -18.156,Z -36.676,A -90.000,B 90.000,C 0.000} C_DIS
LIN {X -107.977,Y -18.146,Z -36.582,A -90.000,B 90.000,C 0.000} C_DIS
LIN {X -107.811,Y -18.143,Z -36.492,A -90.000,B 90.000,C 0.000} C_DIS
LIN {X -107.482,Y -18.124,Z -36.334,A -90.000,B 90.000,C 0.000} C_DIS
LIN {X -107.150,Y -18.100,Z -36.184,A -90.000,B 90.000,C 0.000} C_DIS
LIN {X -107.053,Y -18.094,Z -36.145,A -90.000,B 90.000,C 0.000} C_DIS
LIN {X -106.907,Y -18.091,Z -36.093,A -90.000,B 90.000,C 0.000} C_DIS
LIN {X -106.602,Y -18.173,Z -35.921,A -90.000,B 90.000,C 0.000} C_DIS
LIN {X -106.314,Y -18.263,Z -35.774,A -90.000,B 90.000,C 0.000} C_DIS
LIN {X -106.210,Y -18.295,Z -35.727,A -90.000,B 90.000,C 0.000} C_DIS
LIN {X -106.090,Y -18.333,Z -35.678,A -90.000,B 90.000,C 0.000} C_DIS
LIN {X -105.949,Y -18.331,Z -35.494,A -90.000,B 90.000,C 0.000} C_DIS
LIN {X -105.624,Y -18.333,Z -35.090,A -90.000,B 90.000,C 0.000} C_DIS
LIN {X -105.489,Y -18.325,Z -34.937,A -90.000,B 90.000,C 0.000} C_DIS
LIN {X -105.392,Y -18.320,Z -34.831,A -90.000,B 90.000,C 0.000} C_DIS
LIN {X -105.311,Y -18.317,Z -34.748,A -90.000,B 90.000,C 0.000} C_DIS
LIN {X -105.179,Y -18.316,Z -34.621,A -90.000,B 90.000,C 0.000} C_DIS
LIN {X -104.915,Y -18.319,Z -34.384,A -90.000,B 90.000,C 0.000} C_DIS
LIN {X -104.476,Y -18.300,Z -34.015,A -90.000,B 90.000,C 0.000} C_DIS
LIN {X -104.368,Y -18.298,Z -33.930,A -90.000,B 90.000,C 0.000} C_DIS
LIN {X -104.102,Y -18.297,Z -33.735,A -90.000,B 90.000,C 0.000} C_DIS
LIN {X -103.484,Y -18.285,Z -33.308,A -90.000,B 90.000,C 0.000} C_DIS
LIN {X -103.371,Y -18.283,Z -33.234,A -90.000,B 90.000,C 0.000} C_DIS
LIN {X -102.699,Y -18.285,Z -32.822,A -90.000,B 90.000,C 0.000} C_DIS
LIN {X -102.221,Y -18.291,Z -32.549,A -90.000,B 90.000,C 0.000} C_DIS
LIN {X -101.970,Y -18.292,Z -32.406,A -90.000,B 90.000,C 0.000} C_DIS
LIN {X -101.860,Y -18.293,Z -32.346,A -90.000,B 90.000,C 0.000} C_DIS
LIN {X -101.568,Y -18.293,Z -32.189,A -90.000,B 90.000,C 0.000} C_DIS
LIN {X -101.134,Y -18.287,Z -31.960,A -90.000,B 90.000,C 0.000} C_DIS
LIN {X -100.998,Y -18.286,Z -31.889,A -90.000,B 90.000,C 0.000} C_DIS
LIN {X -100.518,Y -18.268,Z -31.652,A -90.000,B 90.000,C 0.000} C_DIS
LIN {X -100.420,Y -18.267,Z -31.605,A -90.000,B 90.000,C 0.000} C_DIS
LIN {X -100.096,Y -18.255,Z -31.455,A -90.000,B 90.000,C 0.000} C_DIS
LIN {X -99.868,Y -18.244,Z -31.353,A -90.000,B 90.000,C 0.000} C_DIS
LIN {X -99.780,Y -18.241,Z -31.316,A -90.000,B 90.000,C 0.000} C_DIS
LIN {X -99.727,Y -18.193,Z -31.213,A -90.000,B 90.000,C 0.000} C_DIS
LIN {X -99.663,Y -18.140,Z -31.096,A -90.000,B 90.000,C 0.000} C_DIS
LIN {X -99.617,Y -18.144,Z -30.889,A -90.000,B 90.000,C 0.000} C_DIS
LIN {X -99.589,Y -18.150,Z -30.784,A -90.000,B 90.000,C 0.000} C_DIS
LIN {X -99.533,Y -18.163,Z -30.588,A -90.000,B 90.000,C 0.000} C_DIS
LIN {X -99.408,Y -18.168,Z -30.217,A -90.000,B 90.000,C 0.000} C_DIS
LIN {X -99.327,Y -18.162,Z -30.009,A -90.000,B 90.000,C 0.000} C_DIS
LIN {X -99.255,Y -18.162,Z -29.844,A -90.000,B 90.000,C 0.000} C_DIS
LIN {X -99.196,Y -18.162,Z -29.718,A -90.000,B 90.000,C 0.000} C_DIS
LIN {X -99.049,Y -18.169,Z -29.428,A -90.000,B 90.000,C 0.000} C_DIS
LIN {X -98.841,Y -18.160,Z -29.051,A -90.000,B 90.000,C 0.000} C_DIS
LIN {X -98.786,Y -18.160,Z -28.960,A -90.000,B 90.000,C 0.000} C_DIS
LIN {X -98.671,Y -18.159,Z -28.778,A -90.000,B 90.000,C 0.000} C_DIS
LIN {X -98.581,Y -18.161,Z -28.641,A -90.000,B 90.000,C 0.000} C_DIS
LIN {X -98.272,Y -18.155,Z -28.183,A -90.000,B 90.000,C 0.000} C_DIS
LIN {X -98.213,Y -18.153,Z -28.103,A -90.000,B 90.000,C 0.000} C_DIS
LIN {X -97.987,Y -18.150,Z -27.809,A -90.000,B 90.000,C 0.000} C_DIS
LIN {X -97.879,Y -18.146,Z -27.672,A -90.000,B 90.000,C 0.000} C_DIS
LIN {X -97.545,Y -18.143,Z -27.269,A -90.000,B 90.000,C 0.000} C_DIS
LIN {X -97.485,Y -18.143,Z -27.197,A -90.000,B 90.000,C 0.000} C_DIS
LIN {X -97.311,Y -18.139,Z -26.998,A -90.000,B 90.000,C 0.000} C_DIS
LIN {X -97.257,Y -18.139,Z -26.937,A -90.000,B 90.000,C 0.000} C_DIS
LIN {X -97.054,Y -18.134,Z -26.718,A -90.000,B 90.000,C 0.000} C_DIS
LIN {X -97.018,Y -18.133,Z -26.682,A -90.000,B 90.000,C 0.000} C_DIS
LIN {X -96.747,Y -18.133,Z -26.413,A -90.000,B 90.000,C 0.000} C_DIS
LIN {X -96.681,Y -18.135,Z -26.351,A -90.000,B 90.000,C 0.000} C_DIS
LIN {X -96.400,Y -18.135,Z -26.096,A -90.000,B 90.000,C 0.000} C_DIS
LIN {X -96.257,Y -18.127,Z -25.977,A -90.000,B 90.000,C 0.000} C_DIS
LIN {X -96.019,Y -18.116,Z -25.793,A -90.000,B 90.000,C 0.000} C_DIS
LIN {X -95.921,Y -18.114,Z -25.723,A -90.000,B 90.000,C 0.000} C_DIS
LIN {X -95.866,Y -18.111,Z -25.686,A -90.000,B 90.000,C 0.000} C_DIS
LIN {X -95.627,Y -18.093,Z -25.539,A -90.000,B 90.000,C 0.000} C_DIS
LIN {X -95.523,Y -18.087,Z -25.477,A -90.000,B 90.000,C 0.000} C_DIS
LIN {X -95.419,Y -18.077,Z -25.424,A -90.000,B 90.000,C 0.000} C_DIS
LIN {X -95.261,Y -18.061,Z -25.346,A -90.000,B 90.000,C 0.000} C_DIS
LIN {X -95.090,Y -18.047,Z -25.267,A -90.000,B 90.000,C 0.000} C_DIS
LIN {X -94.936,Y -18.037,Z -25.198,A -90.000,B 90.000,C 0.000} C_DIS
LIN {X -94.769,Y -18.014,Z -25.135,A -90.000,B 90.000,C 0.000} C_DIS
LIN {X -94.678,Y -18.005,Z -25.103,A -90.000,B 90.000,C 0.000} C_DIS
LIN {X -94.584,Y -17.999,Z -25.075,A -90.000,B 90.000,C 0.000} C_DIS
LIN {X -94.077,Y -17.940,Z -24.952,A -90.000,B 90.000,C 0.000} C_DIS
LIN {X -94.031,Y -17.935,Z -24.942,A -90.000,B 90.000,C 0.000} C_DIS
LIN {X -93.751,Y -17.892,Z -24.898,A -90.000,B 90.000,C 0.000} C_DIS
LIN {X -93.480,Y -17.851,Z -24.862,A -90.000,B 90.000,C 0.000} C_DIS
LIN {X -93.398,Y -17.840,Z -24.853,A -90.000,B 90.000,C 0.000} C_DIS
LIN {X -93.229,Y -17.821,Z -24.835,A -90.000,B 90.000,C 0.000} C_DIS
LIN {X -92.982,Y -17.786,Z -24.819,A -90.000,B 90.000,C 0.000} C_DIS
LIN {X -92.852,Y -17.771,Z -24.813,A -90.000,B 90.000,C 0.000} C_DIS
LIN {X -92.679,Y -17.745,Z -24.816,A -90.000,B 90.000,C 0.000} C_DIS
LIN {X -92.507,Y -17.720,Z -24.811,A -90.000,B 90.000,C 0.000} C_DIS
LIN {X -92.327,Y -17.693,Z -24.808,A -90.000,B 90.000,C 0.000} C_DIS
LIN {X -92.132,Y -17.666,Z -24.811,A -90.000,B 90.000,C 0.000} C_DIS
LIN {X -92.027,Y -17.653,Z -24.813,A -90.000,B 90.000,C 0.000} C_DIS
LIN {X -91.774,Y -17.627,Z -24.811,A -90.000,B 90.000,C 0.000} C_DIS
LIN {X -91.447,Y -17.591,Z -24.806,A -90.000,B 90.000,C 0.000} C_DIS
LIN {X -91.316,Y -17.571,Z -24.810,A -90.000,B 90.000,C 0.000} C_DIS
LIN {X -90.988,Y -17.534,Z -24.803,A -90.000,B 90.000,C 0.000} C_DIS
LIN {X -90.900,Y -17.525,Z -24.802,A -90.000,B 90.000,C 0.000} C_DIS
LIN {X -90.763,Y -17.515,Z -24.793,A -90.000,B 90.000,C 0.000} C_DIS
LIN {X -90.604,Y -17.494,Z -24.787,A -90.000,B 90.000,C 0.000} C_DIS
LIN {X -90.263,Y -17.458,Z -24.776,A -90.000,B 90.000,C 0.000} C_DIS
LIN {X -90.145,Y -17.449,Z -24.765,A -90.000,B 90.000,C 0.000} C_DIS
LIN {X -89.930,Y -17.429,Z -24.744,A -90.000,B 90.000,C 0.000} C_DIS
LIN {X -89.642,Y -17.400,Z -24.723,A -90.000,B 90.000,C 0.000} C_DIS
LIN {X -89.337,Y -17.376,Z -24.684,A -90.000,B 90.000,C 0.000} C_DIS
LIN {X -89.184,Y -17.369,Z -24.653,A -90.000,B 90.000,C 0.000} C_DIS
LIN {X -88.624,Y -17.339,Z -24.550,A -90.000,B 90.000,C 0.000} C_DIS
LIN {X -88.443,Y -17.331,Z -24.506,A -90.000,B 90.000,C 0.000} C_DIS
LIN {X -88.064,Y -17.322,Z -24.387,A -90.000,B 90.000,C 0.000} C_DIS
LIN {X -87.744,Y -17.317,Z -24.260,A -90.000,B 90.000,C 0.000} C_DIS
LIN {X -87.464,Y -17.314,Z -24.122,A -90.000,B 90.000,C 0.000} C_DIS
LIN {X -87.248,Y -17.313,Z -23.988,A -90.000,B 90.000,C 0.000} C_DIS
LIN {X -87.120,Y -17.314,Z -23.886,A -90.000,B 90.000,C 0.000} C_DIS
LIN {X -87.078,Y -17.314,Z -23.841,A -90.000,B 90.000,C 0.000} C_DIS
LIN {X -86.784,Y -17.322,Z -23.473,A -90.000,B 90.000,C 0.000} C_DIS
LIN {X -86.423,Y -17.331,Z -22.965,A -90.000,B 90.000,C 0.000} C_DIS
LIN {X -86.122,Y -17.333,Z -22.542,A -90.000,B 90.000,C 0.000} C_DIS
LIN {X -86.030,Y -17.333,Z -22.416,A -90.000,B 90.000,C 0.000} C_DIS
LIN {X -85.640,Y -17.334,Z -21.890,A -90.000,B 90.000,C 0.000} C_DIS
LIN {X -85.512,Y -17.335,Z -21.714,A -90.000,B 90.000,C 0.000} C_DIS
LIN {X -85.437,Y -17.337,Z -21.601,A -90.000,B 90.000,C 0.000} C_DIS
LIN {X -85.380,Y -17.352,Z -21.388,A -90.000,B 90.000,C 0.000} C_DIS
LIN {X -85.351,Y -17.362,Z -21.274,A -90.000,B 90.000,C 0.000} C_DIS
LIN {X -85.269,Y -17.390,Z -20.998,A -90.000,B 90.000,C 0.000} C_DIS
LIN {X -85.192,Y -17.420,Z -20.739,A -90.000,B 90.000,C 0.000} C_DIS
LIN {X -85.161,Y -17.432,Z -20.646,A -90.000,B 90.000,C 0.000} C_DIS
LIN {X -85.026,Y -17.458,Z -20.312,A -90.000,B 90.000,C 0.000} C_DIS
LIN {X -84.925,Y -17.472,Z -20.058,A -90.000,B 90.000,C 0.000} C_DIS
LIN {X -84.861,Y -17.480,Z -19.904,A -90.000,B 90.000,C 0.000} C_DIS
LIN {X -84.790,Y -17.484,Z -19.760,A -90.000,B 90.000,C 0.000} C_DIS
LIN {X -84.643,Y -17.496,Z -19.477,A -90.000,B 90.000,C 0.000} C_DIS
LIN {X -84.534,Y -17.501,Z -19.291,A -90.000,B 90.000,C 0.000} C_DIS
LIN {X -84.411,Y -17.512,Z -19.087,A -90.000,B 90.000,C 0.000} C_DIS
LIN {X -84.237,Y -17.519,Z -18.848,A -90.000,B 90.000,C 0.000} C_DIS
LIN {X -84.112,Y -17.526,Z -18.681,A -90.000,B 90.000,C 0.000} C_DIS
LIN {X -83.936,Y -17.540,Z -18.450,A -90.000,B 90.000,C 0.000} C_DIS
LIN {X -83.627,Y -17.549,Z -18.114,A -90.000,B 90.000,C 0.000} C_DIS
LIN {X -83.290,Y -17.547,Z -17.811,A -90.000,B 90.000,C 0.000} C_DIS
LIN {X -83.009,Y -17.557,Z -17.575,A -90.000,B 90.000,C 0.000} C_DIS
LIN {X -82.875,Y -17.559,Z -17.477,A -90.000,B 90.000,C 0.000} C_DIS
LIN {X -82.827,Y -17.561,Z -17.442,A -90.000,B 90.000,C 0.000} C_DIS
LIN {X -82.744,Y -17.567,Z -17.383,A -90.000,B 90.000,C 0.000} C_DIS
LIN {X -82.469,Y -17.573,Z -17.211,A -90.000,B 90.000,C 0.000} C_DIS
LIN {X -82.375,Y -17.576,Z -17.152,A -90.000,B 90.000,C 0.000} C_DIS
LIN {X -82.017,Y -17.583,Z -16.946,A -90.000,B 90.000,C 0.000} C_DIS
LIN {X -81.607,Y -17.592,Z -16.749,A -90.000,B 90.000,C 0.000} C_DIS
LIN {X -81.477,Y -17.595,Z -16.698,A -90.000,B 90.000,C 0.000} C_DIS
LIN {X -80.871,Y -17.610,Z -16.483,A -90.000,B 90.000,C 0.000} C_DIS
LIN {X -80.720,Y -17.614,Z -16.431,A -90.000,B 90.000,C 0.000} C_DIS
LIN {X -80.607,Y -17.612,Z -16.402,A -90.000,B 90.000,C 0.000} C_DIS
LIN {X -80.165,Y -17.621,Z -16.300,A -90.000,B 90.000,C 0.000} C_DIS
LIN {X -80.070,Y -17.622,Z -16.281,A -90.000,B 90.000,C 0.000} C_DIS
LIN {X -79.688,Y -17.634,Z -16.210,A -90.000,B 90.000,C 0.000} C_DIS
LIN {X -79.352,Y -17.637,Z -16.168,A -90.000,B 90.000,C 0.000} C_DIS
LIN {X -79.219,Y -17.640,Z -16.153,A -90.000,B 90.000,C 0.000} C_DIS
LIN {X -79.053,Y -17.641,Z -16.142,A -90.000,B 90.000,C 0.000} C_DIS
LIN {X -78.864,Y -17.645,Z -16.132,A -90.000,B 90.000,C 0.000} C_DIS
LIN {X -78.620,Y -17.652,Z -16.121,A -90.000,B 90.000,C 0.000} C_DIS
LIN {X -78.495,Y -17.656,Z -16.117,A -90.000,B 90.000,C 0.000} C_DIS
LIN {X -78.175,Y -17.659,Z -16.113,A -90.000,B 90.000,C 0.000} C_DIS
LIN {X -78.019,Y -17.658,Z -16.120,A -90.000,B 90.000,C 0.000} C_DIS
LIN {X -77.855,Y -17.658,Z -16.128,A -90.000,B 90.000,C 0.000} C_DIS
LIN {X -77.484,Y -17.666,Z -16.155,A -90.000,B 90.000,C 0.000} C_DIS
LIN {X -77.083,Y -17.679,Z -16.186,A -90.000,B 90.000,C 0.000} C_DIS
LIN {X -76.775,Y -17.675,Z -16.230,A -90.000,B 90.000,C 0.000} C_DIS
LIN {X -76.609,Y -17.674,Z -16.259,A -90.000,B 90.000,C 0.000} C_DIS
LIN {X -76.246,Y -17.679,Z -16.330,A -90.000,B 90.000,C 0.000} C_DIS
LIN {X -75.947,Y -17.687,Z -16.392,A -90.000,B 90.000,C 0.000} C_DIS
LIN {X -75.711,Y -17.696,Z -16.442,A -90.000,B 90.000,C 0.000} C_DIS
LIN {X -75.492,Y -17.700,Z -16.495,A -90.000,B 90.000,C 0.000} C_DIS
LIN {X -75.297,Y -17.697,Z -16.551,A -90.000,B 90.000,C 0.000} C_DIS
LIN {X -75.218,Y -17.697,Z -16.576,A -90.000,B 90.000,C 0.000} C_DIS
LIN {X -74.843,Y -17.704,Z -16.695,A -90.000,B 90.000,C 0.000} C_DIS
LIN {X -74.260,Y -17.726,Z -16.889,A -90.000,B 90.000,C 0.000} C_DIS
LIN {X -74.193,Y -17.727,Z -16.913,A -90.000,B 90.000,C 0.000} C_DIS
LIN {X -73.754,Y -17.724,Z -17.088,A -90.000,B 90.000,C 0.000} C_DIS
LIN {X -73.172,Y -17.734,Z -17.355,A -90.000,B 90.000,C 0.000} C_DIS
LIN {X -72.629,Y -17.746,Z -17.606,A -90.000,B 90.000,C 0.000} C_DIS
LIN {X -72.240,Y -17.738,Z -17.809,A -90.000,B 90.000,C 0.000} C_DIS
LIN {X -71.985,Y -17.741,Z -17.949,A -90.000,B 90.000,C 0.000} C_DIS
LIN {X -71.350,Y -17.767,Z -18.300,A -90.000,B 90.000,C 0.000} C_DIS
LIN {X -70.965,Y -17.780,Z -18.517,A -90.000,B 90.000,C 0.000} C_DIS
LIN {X -70.744,Y -17.783,Z -18.650,A -90.000,B 90.000,C 0.000} C_DIS
LIN {X -70.365,Y -17.791,Z -18.900,A -90.000,B 90.000,C 0.000} C_DIS
LIN {X -69.462,Y -17.829,Z -19.518,A -90.000,B 90.000,C 0.000} C_DIS
LIN {X -69.197,Y -17.832,Z -19.710,A -90.000,B 90.000,C 0.000} C_DIS
LIN {X -69.127,Y -17.834,Z -19.763,A -90.000,B 90.000,C 0.000} C_DIS
LIN {X -68.649,Y -17.860,Z -20.132,A -90.000,B 90.000,C 0.000} C_DIS
LIN {X -68.248,Y -17.879,Z -20.445,A -90.000,B 90.000,C 0.000} C_DIS
LIN {X -68.019,Y -17.885,Z -20.630,A -90.000,B 90.000,C 0.000} C_DIS
LIN {X -67.908,Y -17.889,Z -20.722,A -90.000,B 90.000,C 0.000} C_DIS
LIN {X -67.559,Y -17.911,Z -21.029,A -90.000,B 90.000,C 0.000} C_DIS
LIN {X -67.111,Y -17.940,Z -21.442,A -90.000,B 90.000,C 0.000} C_DIS
LIN {X -66.899,Y -17.958,Z -21.644,A -90.000,B 90.000,C 0.000} C_DIS
LIN {X -66.777,Y -17.965,Z -21.766,A -90.000,B 90.000,C 0.000} C_DIS
LIN {X -66.560,Y -17.971,Z -21.994,A -90.000,B 90.000,C 0.000} C_DIS
LIN {X -66.371,Y -17.978,Z -22.197,A -90.000,B 90.000,C 0.000} C_DIS
LIN {X -66.207,Y -17.991,Z -22.383,A -90.000,B 90.000,C 0.000} C_DIS
LIN {X -66.117,Y -18.002,Z -22.491,A -90.000,B 90.000,C 0.000} C_DIS
LIN {X -65.838,Y -18.029,Z -22.860,A -90.000,B 90.000,C 0.000} C_DIS
LIN {X -65.569,Y -18.052,Z -23.237,A -90.000,B 90.000,C 0.000} C_DIS
LIN {X -65.417,Y -18.062,Z -23.455,A -90.000,B 90.000,C 0.000} C_DIS
LIN {X -65.331,Y -18.070,Z -23.585,A -90.000,B 90.000,C 0.000} C_DIS
LIN {X -65.085,Y -18.104,Z -23.976,A -90.000,B 90.000,C 0.000} C_DIS
LIN {X -64.874,Y -18.122,Z -24.330,A -90.000,B 90.000,C 0.000} C_DIS
LIN {X -64.690,Y -18.138,Z -24.673,A -90.000,B 90.000,C 0.000} C_DIS
LIN {X -64.610,Y -18.151,Z -24.818,A -90.000,B 90.000,C 0.000} C_DIS
LIN {X -64.493,Y -18.174,Z -25.045,A -90.000,B 90.000,C 0.000} C_DIS
LIN {X -64.351,Y -18.191,Z -25.340,A -90.000,B 90.000,C 0.000} C_DIS
LIN {X -64.219,Y -18.202,Z -25.622,A -90.000,B 90.000,C 0.000} C_DIS
LIN {X -64.159,Y -18.208,Z -25.751,A -90.000,B 90.000,C 0.000} C_DIS
LIN {X -63.954,Y -18.241,Z -26.233,A -90.000,B 90.000,C 0.000} C_DIS
LIN {X -63.752,Y -18.281,Z -26.700,A -90.000,B 90.000,C 0.000} C_DIS
LIN {X -63.684,Y -18.292,Z -26.862,A -90.000,B 90.000,C 0.000} C_DIS
LIN {X -63.633,Y -18.303,Z -26.996,A -90.000,B 90.000,C 0.000} C_DIS
LIN {X -63.519,Y -18.330,Z -27.311,A -90.000,B 90.000,C 0.000} C_DIS
LIN {X -63.508,Y -18.331,Z -27.335,A -90.000,B 90.000,C 0.000} C_DIS
LIN {X -63.371,Y -18.368,Z -27.596,A -90.000,B 90.000,C 0.000} C_DIS
LIN {X -63.191,Y -18.421,Z -27.952,A -90.000,B 90.000,C 0.000} C_DIS
LIN {X -63.107,Y -18.422,Z -28.054,A -90.000,B 90.000,C 0.000} C_DIS
LIN {X -62.909,Y -18.453,Z -28.271,A -90.000,B 90.000,C 0.000} C_DIS
LIN {X -62.327,Y -18.454,Z -28.680,A -90.000,B 90.000,C 0.000} C_DIS
LIN {X -62.250,Y -18.461,Z -28.730,A -90.000,B 90.000,C 0.000} C_DIS
LIN {X -62.229,Y -18.461,Z -28.740,A -90.000,B 90.000,C 0.000} C_DIS
LIN {X -61.763,Y -18.465,Z -28.956,A -90.000,B 90.000,C 0.000} C_DIS
LIN {X -61.190,Y -18.473,Z -29.220,A -90.000,B 90.000,C 0.000} C_DIS
LIN {X -61.036,Y -18.480,Z -29.288,A -90.000,B 90.000,C 0.000} C_DIS
LIN {X -60.552,Y -18.485,Z -29.461,A -90.000,B 90.000,C 0.000} C_DIS
LIN {X -59.478,Y -18.508,Z -29.838,A -90.000,B 90.000,C 0.000} C_DIS
LIN {X -59.367,Y -18.510,Z -29.873,A -90.000,B 90.000,C 0.000} C_DIS
LIN {X -58.995,Y -18.514,Z -29.980,A -90.000,B 90.000,C 0.000} C_DIS
LIN {X -57.906,Y -18.530,Z -30.302,A -90.000,B 90.000,C 0.000} C_DIS
LIN {X -57.562,Y -18.537,Z -30.410,A -90.000,B 90.000,C 0.000} C_DIS
LIN {X -57.223,Y -18.549,Z -30.515,A -90.000,B 90.000,C 0.000} C_DIS
LIN {X -56.003,Y -18.560,Z -30.814,A -90.000,B 90.000,C 0.000} C_DIS
LIN {X -55.260,Y -18.565,Z -30.990,A -90.000,B 90.000,C 0.000} C_DIS
LIN {X -55.183,Y -18.567,Z -31.008,A -90.000,B 90.000,C 0.000} C_DIS
LIN {X -53.934,Y -18.569,Z -31.195,A -90.000,B 90.000,C 0.000} C_DIS
LIN {X -52.693,Y -18.558,Z -31.386,A -90.000,B 90.000,C 0.000} C_DIS
LIN {X -52.543,Y -18.551,Z -31.396,A -90.000,B 90.000,C 0.000} C_DIS
LIN {X -51.345,Y -18.527,Z -31.459,A -90.000,B 90.000,C 0.000} C_DIS
LIN {X -51.119,Y -18.517,Z -31.475,A -90.000,B 90.000,C 0.000} C_DIS
LIN {X -50.769,Y -18.504,Z -31.505,A -90.000,B 90.000,C 0.000} C_DIS
LIN {X -50.393,Y -18.492,Z -31.541,A -90.000,B 90.000,C 0.000} C_DIS
LIN {X -50.041,Y -18.476,Z -31.578,A -90.000,B 90.000,C 0.000} C_DIS
LIN {X -49.812,Y -18.472,Z -31.597,A -90.000,B 90.000,C 0.000} C_DIS
LIN {X -49.601,Y -18.466,Z -31.610,A -90.000,B 90.000,C 0.000} C_DIS
LIN {X -49.306,Y -18.442,Z -31.587,A -90.000,B 90.000,C 0.000} C_DIS
LIN {X -49.122,Y -18.431,Z -31.581,A -90.000,B 90.000,C 0.000} C_DIS
LIN {X -48.332,Y -18.402,Z -31.589,A -90.000,B 90.000,C 0.000} C_DIS
LIN {X -48.201,Y -18.399,Z -31.594,A -90.000,B 90.000,C 0.000} C_DIS
LIN {X -47.849,Y -18.397,Z -31.618,A -90.000,B 90.000,C 0.000} C_DIS
LIN {X -46.684,Y -18.377,Z -31.704,A -90.000,B 90.000,C 0.000} C_DIS
LIN {X -46.239,Y -18.357,Z -31.715,A -90.000,B 90.000,C 0.000} C_DIS
LIN {X -45.587,Y -18.343,Z -31.724,A -90.000,B 90.000,C 0.000} C_DIS
LIN {X -45.507,Y -18.342,Z -31.726,A -90.000,B 90.000,C 0.000} C_DIS
LIN {X -45.074,Y -18.341,Z -31.747,A -90.000,B 90.000,C 0.000} C_DIS
LIN {X -42.913,Y -18.313,Z -31.863,A -90.000,B 90.000,C 0.000} C_DIS
LIN {X -42.597,Y -18.304,Z -31.871,A -90.000,B 90.000,C 0.000} C_DIS
LIN {X -42.230,Y -18.298,Z -31.879,A -90.000,B 90.000,C 0.000} C_DIS
LIN {X -41.541,Y -18.290,Z -31.899,A -90.000,B 90.000,C 0.000} C_DIS
LIN {X -41.220,Y -18.283,Z -31.913,A -90.000,B 90.000,C 0.000} C_DIS
LIN {X -39.165,Y -18.252,Z -32.029,A -90.000,B 90.000,C 0.000} C_DIS
LIN {X -38.605,Y -18.239,Z -32.055,A -90.000,B 90.000,C 0.000} C_DIS
LIN {X -37.287,Y -18.215,Z -32.116,A -90.000,B 90.000,C 0.000} C_DIS
LIN {X -36.282,Y -18.214,Z -32.192,A -90.000,B 90.000,C 0.000} C_DIS
LIN {X -34.891,Y -18.179,Z -32.322,A -90.000,B 90.000,C 0.000} C_DIS
LIN {X -32.292,Y -18.111,Z -32.580,A -90.000,B 90.000,C 0.000} C_DIS
LIN {X -31.977,Y -18.103,Z -32.618,A -90.000,B 90.000,C 0.000} C_DIS
LIN {X -30.791,Y -18.083,Z -32.778,A -90.000,B 90.000,C 0.000} C_DIS
LIN {X -30.510,Y -18.081,Z -32.820,A -90.000,B 90.000,C 0.000} C_DIS
LIN {X -29.473,Y -18.060,Z -32.985,A -90.000,B 90.000,C 0.000} C_DIS
LIN {X -28.905,Y -18.046,Z -33.069,A -90.000,B 90.000,C 0.000} C_DIS
LIN {X -28.440,Y -18.037,Z -33.136,A -90.000,B 90.000,C 0.000} C_DIS
LIN {X -27.647,Y -18.026,Z -33.260,A -90.000,B 90.000,C 0.000} C_DIS
LIN {X -27.255,Y -18.019,Z -33.322,A -90.000,B 90.000,C 0.000} C_DIS
LIN {X -27.004,Y -18.012,Z -33.357,A -90.000,B 90.000,C 0.000} C_DIS
LIN {X -26.258,Y -17.996,Z -33.457,A -90.000,B 90.000,C 0.000} C_DIS
LIN {X -25.667,Y -17.976,Z -33.544,A -90.000,B 90.000,C 0.000} C_DIS
LIN {X -24.738,Y -17.965,Z -33.701,A -90.000,B 90.000,C 0.000} C_DIS
LIN {X -22.841,Y -17.935,Z -34.020,A -90.000,B 90.000,C 0.000} C_DIS
LIN {X -21.039,Y -17.901,Z -34.322,A -90.000,B 90.000,C 0.000} C_DIS
LIN {X -20.478,Y -17.885,Z -34.422,A -90.000,B 90.000,C 0.000} C_DIS
LIN {X -19.300,Y -17.856,Z -34.651,A -90.000,B 90.000,C 0.000} C_DIS
LIN {X -17.667,Y -17.846,Z -34.998,A -90.000,B 90.000,C 0.000} C_DIS
LIN {X -17.391,Y -17.844,Z -35.063,A -90.000,B 90.000,C 0.000} C_DIS
LIN {X -16.214,Y -17.846,Z -35.332,A -90.000,B 90.000,C 0.000} C_DIS
LIN {X -15.198,Y -17.856,Z -35.553,A -90.000,B 90.000,C 0.000} C_DIS
LIN {X -14.814,Y -17.853,Z -35.647,A -90.000,B 90.000,C 0.000} C_DIS
LIN {X -13.261,Y -17.860,Z -36.050,A -90.000,B 90.000,C 0.000} C_DIS
LIN {X -12.921,Y -17.866,Z -36.134,A -90.000,B 90.000,C 0.000} C_DIS
LIN {X -12.212,Y -17.881,Z -36.317,A -90.000,B 90.000,C 0.000} C_DIS
LIN {X -11.688,Y -17.883,Z -36.459,A -90.000,B 90.000,C 0.000} C_DIS
LIN {X -11.468,Y -17.888,Z -36.516,A -90.000,B 90.000,C 0.000} C_DIS
LIN {X -9.474,Y -17.954,Z -37.061,A -90.000,B 90.000,C 0.000} C_DIS
LIN {X -8.227,Y -18.011,Z -37.390,A -90.000,B 90.000,C 0.000} C_DIS
LIN {X -7.974,Y -18.026,Z -37.462,A -90.000,B 90.000,C 0.000} C_DIS
LIN {X -6.696,Y -18.118,Z -37.812,A -90.000,B 90.000,C 0.000} C_DIS
LIN {X -6.481,Y -18.133,Z -37.870,A -90.000,B 90.000,C 0.000} C_DIS
LIN {X -6.229,Y -18.147,Z -37.939,A -90.000,B 90.000,C 0.000} C_DIS
LIN {X -5.067,Y -18.233,Z -38.251,A -90.000,B 90.000,C 0.000} C_DIS
LIN {X -4.773,Y -18.258,Z -38.335,A -90.000,B 90.000,C 0.000} C_DIS
LIN {X -3.964,Y -18.307,Z -38.541,A -90.000,B 90.000,C 0.000} C_DIS
LIN {X -3.524,Y -18.344,Z -38.648,A -90.000,B 90.000,C 0.000} C_DIS
LIN {X -3.060,Y -18.372,Z -38.738,A -90.000,B 90.000,C 0.000} C_DIS
LIN {X -2.374,Y -18.405,Z -38.853,A -90.000,B 90.000,C 0.000} C_DIS
LIN {X -1.557,Y -18.414,Z -38.942,A -90.000,B 90.000,C 0.000} C_DIS
LIN {X -1.372,Y -18.415,Z -38.963,A -90.000,B 90.000,C 0.000} C_DIS
LIN {X -1.133,Y -18.422,Z -38.987,A -90.000,B 90.000,C 0.000} C_DIS
LIN {X -0.625,Y -18.422,Z -39.010,A -90.000,B 90.000,C 0.000} C_DIS
LIN {X 0.450,Y -18.414,Z -39.065,A -90.000,B 90.000,C 0.000} C_DIS
LIN {X 1.000,Y -18.412,Z -39.098,A -90.000,B 90.000,C 0.000} C_DIS
LIN {X 3.290,Y -18.351,Z -39.180,A -90.000,B 90.000,C 0.000} C_DIS
LIN {X 3.831,Y -18.334,Z -39.196,A -90.000,B 90.000,C 0.000} C_DIS
LIN {X 5.483,Y -18.273,Z -39.250,A -90.000,B 90.000,C 0.000} C_DIS
LIN {X 5.669,Y -18.266,Z -39.254,A -90.000,B 90.000,C 0.000} C_DIS
LIN {X 6.032,Y -18.257,Z -39.267,A -90.000,B 90.000,C 0.000} C_DIS
LIN {X 6.320,Y -18.250,Z -39.279,A -90.000,B 90.000,C 0.000} C_DIS
LIN {X 7.547,Y -18.200,Z -39.347,A -90.000,B 90.000,C 0.000} C_DIS
LIN {X 7.845,Y -18.187,Z -39.366,A -90.000,B 90.000,C 0.000} C_DIS
LIN {X 8.088,Y -18.180,Z -39.389,A -90.000,B 90.000,C 0.000} C_DIS
LIN {X 8.639,Y -18.163,Z -39.434,A -90.000,B 90.000,C 0.000} C_DIS
LIN {X 8.697,Y -18.162,Z -39.438,A -90.000,B 90.000,C 0.000} C_DIS
LIN {X 9.530,Y -18.135,Z -39.509,A -90.000,B 90.000,C 0.000} C_DIS
LIN {X 10.413,Y -18.091,Z -39.595,A -90.000,B 90.000,C 0.000} C_DIS
LIN {X 10.828,Y -18.075,Z -39.642,A -90.000,B 90.000,C 0.000} C_DIS
LIN {X 11.284,Y -18.055,Z -39.691,A -90.000,B 90.000,C 0.000} C_DIS
LIN {X 11.967,Y -18.031,Z -39.760,A -90.000,B 90.000,C 0.000} C_DIS
LIN {X 13.788,Y -17.951,Z -39.959,A -90.000,B 90.000,C 0.000} C_DIS
LIN {X 14.338,Y -17.933,Z -40.014,A -90.000,B 90.000,C 0.000} C_DIS
LIN {X 15.419,Y -17.904,Z -40.116,A -90.000,B 90.000,C 0.000} C_DIS
LIN {X 16.088,Y -17.881,Z -40.174,A -90.000,B 90.000,C 0.000} C_DIS
LIN {X 17.559,Y -17.884,Z -40.237,A -90.000,B 90.000,C 0.000} C_DIS
LIN {X 18.544,Y -17.867,Z -40.267,A -90.000,B 90.000,C 0.000} C_DIS
LIN {X 18.752,Y -17.870,Z -40.267,A -90.000,B 90.000,C 0.000} C_DIS
LIN {X 19.969,Y -17.909,Z -40.241,A -90.000,B 90.000,C 0.000} C_DIS
LIN {X 21.249,Y -17.911,Z -40.179,A -90.000,B 90.000,C 0.000} C_DIS
LIN {X 21.797,Y -17.922,Z -40.143,A -90.000,B 90.000,C 0.000} C_DIS
LIN {X 22.051,Y -17.929,Z -40.125,A -90.000,B 90.000,C 0.000} C_DIS
LIN {X 22.866,Y -17.928,Z -40.044,A -90.000,B 90.000,C 0.000} C_DIS
LIN {X 23.110,Y -17.925,Z -40.016,A -90.000,B 90.000,C 0.000} C_DIS
LIN {X 23.979,Y -17.922,Z -39.907,A -90.000,B 90.000,C 0.000} C_DIS
LIN {X 24.831,Y -17.896,Z -39.775,A -90.000,B 90.000,C 0.000} C_DIS
LIN {X 25.006,Y -17.892,Z -39.749,A -90.000,B 90.000,C 0.000} C_DIS
LIN {X 25.282,Y -17.889,Z -39.704,A -90.000,B 90.000,C 0.000} C_DIS
LIN {X 25.747,Y -17.882,Z -39.630,A -90.000,B 90.000,C 0.000} C_DIS
LIN {X 26.087,Y -17.866,Z -39.565,A -90.000,B 90.000,C 0.000} C_DIS
LIN {X 26.846,Y -17.835,Z -39.430,A -90.000,B 90.000,C 0.000} C_DIS
LIN {X 27.389,Y -17.821,Z -39.323,A -90.000,B 90.000,C 0.000} C_DIS
LIN {X 27.742,Y -17.820,Z -39.259,A -90.000,B 90.000,C 0.000} C_DIS
LIN {X 27.792,Y -17.819,Z -39.251,A -90.000,B 90.000,C 0.000} C_DIS
LIN {X 28.123,Y -17.800,Z -39.188,A -90.000,B 90.000,C 0.000} C_DIS
LIN {X 28.745,Y -17.758,Z -39.079,A -90.000,B 90.000,C 0.000} C_DIS
LIN {X 28.804,Y -17.756,Z -39.069,A -90.000,B 90.000,C 0.000} C_DIS
LIN {X 29.010,Y -17.755,Z -39.028,A -90.000,B 90.000,C 0.000} C_DIS
LIN {X 29.534,Y -17.744,Z -38.934,A -90.000,B 90.000,C 0.000} C_DIS
LIN {X 29.882,Y -17.732,Z -38.878,A -90.000,B 90.000,C 0.000} C_DIS
LIN {X 30.190,Y -17.711,Z -38.822,A -90.000,B 90.000,C 0.000} C_DIS
LIN {X 30.638,Y -17.692,Z -38.751,A -90.000,B 90.000,C 0.000} C_DIS
LIN {X 30.773,Y -17.686,Z -38.730,A -90.000,B 90.000,C 0.000} C_DIS
LIN {X 31.087,Y -17.665,Z -38.692,A -90.000,B 90.000,C 0.000} C_DIS
LIN {X 31.700,Y -17.641,Z -38.599,A -90.000,B 90.000,C 0.000} C_DIS
LIN {X 32.115,Y -17.630,Z -38.540,A -90.000,B 90.000,C 0.000} C_DIS
LIN {X 32.506,Y -17.627,Z -38.491,A -90.000,B 90.000,C 0.000} C_DIS
LIN {X 32.665,Y -17.620,Z -38.469,A -90.000,B 90.000,C 0.000} C_DIS
LIN {X 33.453,Y -17.560,Z -38.404,A -90.000,B 90.000,C 0.000} C_DIS
LIN {X 33.675,Y -17.553,Z -38.373,A -90.000,B 90.000,C 0.000} C_DIS
LIN {X 34.081,Y -17.550,Z -38.323,A -90.000,B 90.000,C 0.000} C_DIS
LIN {X 34.618,Y -17.536,Z -38.276,A -90.000,B 90.000,C 0.000} C_DIS
LIN {X 35.448,Y -17.502,Z -38.232,A -90.000,B 90.000,C 0.000} C_DIS
LIN {X 35.735,Y -17.491,Z -38.217,A -90.000,B 90.000,C 0.000} C_DIS
LIN {X 35.935,Y -17.486,Z -38.208,A -90.000,B 90.000,C 0.000} C_DIS
LIN {X 36.641,Y -17.464,Z -38.193,A -90.000,B 90.000,C 0.000} C_DIS
LIN {X 37.099,Y -17.449,Z -38.193,A -90.000,B 90.000,C 0.000} C_DIS
LIN {X 37.827,Y -17.419,Z -38.218,A -90.000,B 90.000,C 0.000} C_DIS
LIN {X 38.294,Y -17.411,Z -38.238,A -90.000,B 90.000,C 0.000} C_DIS
LIN {X 39.608,Y -17.385,Z -38.324,A -90.000,B 90.000,C 0.000} C_DIS
LIN {X 39.988,Y -17.370,Z -38.379,A -90.000,B 90.000,C 0.000} C_DIS
LIN {X 40.461,Y -17.359,Z -38.450,A -90.000,B 90.000,C 0.000} C_DIS
LIN {X 42.208,Y -17.336,Z -38.714,A -90.000,B 90.000,C 0.000} C_DIS
LIN {X 42.559,Y -17.335,Z -38.764,A -90.000,B 90.000,C 0.000} C_DIS
LIN {X 43.031,Y -17.333,Z -38.852,A -90.000,B 90.000,C 0.000} C_DIS
LIN {X 44.058,Y -17.325,Z -39.108,A -90.000,B 90.000,C 0.000} C_DIS
LIN {X 44.158,Y -17.325,Z -39.133,A -90.000,B 90.000,C 0.000} C_DIS
LIN {X 45.241,Y -17.317,Z -39.452,A -90.000,B 90.000,C 0.000} C_DIS
LIN {X 45.816,Y -17.315,Z -39.623,A -90.000,B 90.000,C 0.000} C_DIS
LIN {X 46.386,Y -17.315,Z -39.803,A -90.000,B 90.000,C 0.000} C_DIS
LIN {X 47.404,Y -17.311,Z -40.226,A -90.000,B 90.000,C 0.000} C_DIS
LIN {X 48.322,Y -17.310,Z -40.608,A -90.000,B 90.000,C 0.000} C_DIS
LIN {X 49.484,Y -17.309,Z -41.114,A -90.000,B 90.000,C 0.000} C_DIS
LIN {X 49.658,Y -17.309,Z -41.202,A -90.000,B 90.000,C 0.000} C_DIS
LIN {X 50.074,Y -17.309,Z -41.422,A -90.000,B 90.000,C 0.000} C_DIS
LIN {X 50.675,Y -17.332,Z -41.740,A -90.000,B 90.000,C 0.000} C_DIS
LIN {X 52.060,Y -17.308,Z -42.475,A -90.000,B 90.000,C 0.000} C_DIS
LIN {X 52.264,Y -19.982,Z -42.583,A -90.000,B 90.000,C 0.000} C_DIS
LIN {X 52.290,Y -19.959,Z -42.596,A -90.000,B 90.000,C 0.000} C_DIS
LIN {X 52.294,Y -19.944,Z -42.597,A -90.000,B 90.000,C 0.000} C_DIS
LIN {X 52.323,Y -19.959,Z -42.613,A -90.000,B 90.000,C 0.000} C_DIS
LIN {X 52.524,Y -17.308,Z -42.726,A -90.000,B 90.000,C 0.000} C_DIS
LIN {X 52.699,Y -17.308,Z -42.823,A -90.000,B 90.000,C 0.000} C_DIS
LIN {X 52.743,Y -17.308,Z -42.848,A -90.000,B 90.000,C 0.000} C_DIS
LIN {X 52.798,Y -17.308,Z -42.886,A -90.000,B 90.000,C 0.000} C_DIS
LIN {X 54.038,Y -17.308,Z -43.668,A -90.000,B 90.000,C 0.000} C_DIS
LIN {X 54.463,Y -17.308,Z -43.931,A -90.000,B 90.000,C 0.000} C_DIS
LIN {X 54.573,Y -17.308,Z -43.994,A -90.000,B 90.000,C 0.000} C_DIS
LIN {X 54.595,Y -17.308,Z -44.005,A -90.000,B 90.000,C 0.000} C_DIS
LIN {X 54.604,Y -17.308,Z -44.008,A -90.000,B 90.000,C 0.000} C_DIS
LIN {X 54.608,Y -17.308,Z -44.006,A -90.000,B 90.000,C 0.000} C_DIS
LIN {X 54.616,Y -17.308,Z -44.010,A -90.000,B 90.000,C 0.000} C_DIS
LIN {X 55.155,Y -17.308,Z -44.374,A -90.000,B 90.000,C 0.000} C_DIS
LIN {X 55.508,Y -17.308,Z -44.614,A -90.000,B 90.000,C 0.000} C_DIS
LIN {X 55.664,Y -17.306,Z -44.722,A -90.000,B 90.000,C 0.000} C_DIS
LIN {X 55.668,Y -17.305,Z -44.728,A -90.000,B 90.000,C 0.000} C_DIS
LIN {X 55.684,Y -17.305,Z -44.742,A -90.000,B 90.000,C 0.000} C_DIS
LIN {X 55.818,Y -17.308,Z -44.844,A -90.000,B 90.000,C 0.000} C_DIS
LIN {X 56.414,Y -17.325,Z -45.286,A -90.000,B 90.000,C 0.000} C_DIS
LIN {X 57.697,Y -17.308,Z -46.238,A -90.000,B 90.000,C 0.000} C_DIS
LIN {X 57.986,Y -17.286,Z -46.453,A -90.000,B 90.000,C 0.000} C_DIS
LIN {X 58.139,Y -17.240,Z -46.568,A -90.000,B 90.000,C 0.000} C_DIS
LIN {X 58.178,Y -17.213,Z -46.598,A -90.000,B 90.000,C 0.000} C_DIS
LIN {X 58.199,Y -17.185,Z -46.617,A -90.000,B 90.000,C 0.000} C_DIS
LIN {X 58.208,Y -17.158,Z -46.627,A -90.000,B 90.000,C 0.000} C_DIS
LIN {X 58.212,Y -17.118,Z -46.638,A -90.000,B 90.000,C 0.000} C_DIS
LIN {X 58.217,Y -17.108,Z -46.649,A -90.000,B 90.000,C 0.000} C_DIS
LIN {X 58.232,Y -17.107,Z -46.667,A -90.000,B 90.000,C 0.000} C_DIS
LIN {X 58.262,Y -17.117,Z -46.698,A -90.000,B 90.000,C 0.000} C_DIS
LIN {X 58.312,Y -17.141,Z -46.746,A -90.000,B 90.000,C 0.000} C_DIS
LIN {X 58.499,Y -17.234,Z -46.905,A -90.000,B 90.000,C 0.000} C_DIS
LIN {X 58.639,Y -17.308,Z -47.032,A -90.000,B 90.000,C 0.000} C_DIS
LIN {X 58.681,Y -17.330,Z -47.067,A -90.000,B 90.000,C 0.000} C_DIS
LIN {X 60.135,Y -17.308,Z -48.298,A -90.000,B 90.000,C 0.000} C_DIS
LIN {X 61.125,Y -17.309,Z -49.132,A -90.000,B 90.000,C 0.000} C_DIS
LIN {X 61.658,Y -17.310,Z -49.564,A -90.000,B 90.000,C 0.000} C_DIS
LIN {X 62.534,Y -17.313,Z -50.215,A -90.000,B 90.000,C 0.000} C_DIS
LIN {X 63.430,Y -17.318,Z -50.888,A -90.000,B 90.000,C 0.000} C_DIS
LIN {X 63.519,Y -17.319,Z -50.957,A -90.000,B 90.000,C 0.000} C_DIS
LIN {X 64.865,Y -17.330,Z -51.832,A -90.000,B 90.000,C 0.000} C_DIS
LIN {X 65.231,Y -17.333,Z -52.070,A -90.000,B 90.000,C 0.000} C_DIS
LIN {X 65.675,Y -17.336,Z -52.335,A -90.000,B 90.000,C 0.000} C_DIS
LIN {X 66.707,Y -17.342,Z -52.918,A -90.000,B 90.000,C 0.000} C_DIS
LIN {X 67.279,Y -17.344,Z -53.244,A -90.000,B 90.000,C 0.000} C_DIS
LIN {X 67.589,Y -17.345,Z -53.416,A -90.000,B 90.000,C 0.000} C_DIS
LIN {X 69.001,Y -17.347,Z -54.215,A -90.000,B 90.000,C 0.000} C_DIS
LIN {X 69.725,Y -17.349,Z -54.621,A -90.000,B 90.000,C 0.000} C_DIS
LIN {X 71.799,Y -17.349,Z -55.854,A -90.000,B 90.000,C 0.000} C_DIS
LIN {X 71.925,Y -17.350,Z -55.930,A -90.000,B 90.000,C 0.000} C_DIS
LIN {X 74.096,Y -17.350,Z -57.359,A -90.000,B 90.000,C 0.000} C_DIS
LIN {X 74.354,Y -17.353,Z -57.531,A -90.000,B 90.000,C 0.000} C_DIS
LIN {X 74.569,Y -17.354,Z -57.699,A -90.000,B 90.000,C 0.000} C_DIS
LIN {X 76.096,Y -17.360,Z -58.867,A -90.000,B 90.000,C 0.000} C_DIS
LIN {X 76.368,Y -17.360,Z -59.092,A -90.000,B 90.000,C 0.000} C_DIS
LIN {X 76.485,Y -17.362,Z -59.189,A -90.000,B 90.000,C 0.000} C_DIS
LIN {X 77.314,Y -17.369,Z -59.923,A -90.000,B 90.000,C 0.000} C_DIS
LIN {X 77.887,Y -17.371,Z -60.428,A -90.000,B 90.000,C 0.000} C_DIS
LIN {X 77.928,Y -17.372,Z -60.464,A -90.000,B 90.000,C 0.000} C_DIS
LIN {X 77.928,Y -60.000,Z -60.464,A -90.000,B 90.000,C 0.000} C_DIS
LIN {X 93.909,Y -60.000,Z -42.337,A -90.000,B 90.000,C 0.000} C_DIS
LIN {X 93.909,Y -17.308,Z -42.337,A -90.000,B 90.000,C 0.000} C_DIS
LIN {X 94.433,Y -17.308,Z -42.006,A -90.000,B 90.000,C 0.000} C_DIS
LIN {X 94.958,Y -17.308,Z -41.667,A -90.000,B 90.000,C 0.000} C_DIS
LIN {X 95.088,Y -17.308,Z -41.577,A -90.000,B 90.000,C 0.000} C_DIS
LIN {X 95.112,Y -17.308,Z -41.558,A -90.000,B 90.000,C 0.000} C_DIS
LIN {X 95.120,Y -17.308,Z -41.549,A -90.000,B 90.000,C 0.000} C_DIS
LIN {X 95.121,Y -17.308,Z -41.544,A -90.000,B 90.000,C 0.000} C_DIS
LIN {X 95.130,Y -17.308,Z -41.538,A -90.000,B 90.000,C 0.000} C_DIS
LIN {X 95.838,Y -17.308,Z -41.136,A -90.000,B 90.000,C 0.000} C_DIS
LIN {X 95.969,Y -17.308,Z -41.061,A -90.000,B 90.000,C 0.000} C_DIS
LIN {X 96.484,Y -17.308,Z -40.757,A -90.000,B 90.000,C 0.000} C_DIS
LIN {X 96.937,Y -17.307,Z -40.497,A -90.000,B 90.000,C 0.000} C_DIS
LIN {X 97.333,Y -17.308,Z -40.276,A -90.000,B 90.000,C 0.000} C_DIS
LIN {X 97.952,Y -17.308,Z -39.912,A -90.000,B 90.000,C 0.000} C_DIS
LIN {X 98.534,Y -17.308,Z -39.559,A -90.000,B 90.000,C 0.000} C_DIS
LIN {X 98.742,Y -17.308,Z -39.427,A -90.000,B 90.000,C 0.000} C_DIS
LIN {X 98.891,Y -17.308,Z -39.323,A -90.000,B 90.000,C 0.000} C_DIS
LIN {X 98.902,Y -17.308,Z -39.326,A -90.000,B 90.000,C 0.000} C_DIS
LIN {X 98.951,Y -17.308,Z -39.319,A -90.000,B 90.000,C 0.000} C_DIS
LIN {X 99.074,Y -17.308,Z -39.282,A -90.000,B 90.000,C 0.000} C_DIS
LIN {X 99.306,Y -17.308,Z -39.197,A -90.000,B 90.000,C 0.000} C_DIS
LIN {X 99.684,Y -17.308,Z -39.048,A -90.000,B 90.000,C 0.000} C_DIS
LIN {X 100.241,Y -17.308,Z -38.815,A -90.000,B 90.000,C 0.000} C_DIS
LIN {X 100.599,Y -17.308,Z -38.661,A -90.000,B 90.000,C 0.000} C_DIS
LIN {X 101.014,Y -17.308,Z -38.480,A -90.000,B 90.000,C 0.000} C_DIS
LIN {X 101.487,Y -17.307,Z -38.257,A -90.000,B 90.000,C 0.000} C_DIS
LIN {X 102.038,Y -17.308,Z -38.027,A -90.000,B 90.000,C 0.000} C_DIS
LIN {X 102.165,Y -17.308,Z -37.970,A -90.000,B 90.000,C 0.000} C_DIS
LIN {X 102.630,Y -33.353,Z -37.762,A -90.000,B 90.000,C 0.000} C_DIS
LIN {X 102.687,Y -33.364,Z -37.735,A -90.000,B 90.000,C 0.000} C_DIS
LIN {X 102.695,Y -33.360,Z -37.732,A -90.000,B 90.000,C 0.000} C_DIS
LIN {X 102.697,Y -33.348,Z -37.730,A -90.000,B 90.000,C 0.000} C_DIS
LIN {X 102.704,Y -33.348,Z -37.727,A -90.000,B 90.000,C 0.000} C_DIS
LIN {X 102.762,Y -33.377,Z -37.701,A -90.000,B 90.000,C 0.000} C_DIS
LIN {X 103.228,Y -17.308,Z -37.495,A -90.000,B 90.000,C 0.000} C_DIS
LIN {X 103.365,Y -17.308,Z -37.434,A -90.000,B 90.000,C 0.000} C_DIS
LIN {X 103.550,Y -17.308,Z -37.337,A -90.000,B 90.000,C 0.000} C_DIS
LIN {X 103.734,Y -17.308,Z -37.253,A -90.000,B 90.000,C 0.000} C_DIS
LIN {X 103.917,Y -17.308,Z -37.183,A -90.000,B 90.000,C 0.000} C_DIS
LIN {X 104.257,Y -17.308,Z -37.020,A -90.000,B 90.000,C 0.000} C_DIS
LIN {X 104.724,Y -17.308,Z -36.785,A -90.000,B 90.000,C 0.000} C_DIS
LIN {X 105.145,Y -17.308,Z -36.560,A -90.000,B 90.000,C 0.000} C_DIS
LIN {X 105.520,Y -17.308,Z -36.344,A -90.000,B 90.000,C 0.000} C_DIS
LIN {X 105.853,Y -17.308,Z -36.137,A -90.000,B 90.000,C 0.000} C_DIS
LIN {X 106.147,Y -17.308,Z -35.941,A -90.000,B 90.000,C 0.000} C_DIS
LIN {X 106.322,Y -17.308,Z -35.815,A -90.000,B 90.000,C 0.000} C_DIS
LIN {X 106.482,Y -17.308,Z -35.694,A -90.000,B 90.000,C 0.000} C_DIS
LIN {X 106.693,Y -17.308,Z -35.520,A -90.000,B 90.000,C 0.000} C_DIS
LIN {X 106.816,Y -17.308,Z -35.409,A -90.000,B 90.000,C 0.000} C_DIS
LIN {X 106.927,Y -17.308,Z -35.303,A -90.000,B 90.000,C 0.000} C_DIS
LIN {X 107.025,Y -17.308,Z -35.201,A -90.000,B 90.000,C 0.000} C_DIS
LIN {X 107.112,Y -17.308,Z -35.103,A -90.000,B 90.000,C 0.000} C_DIS
LIN {X 107.188,Y -17.308,Z -35.009,A -90.000,B 90.000,C 0.000} C_DIS
LIN {X 107.254,Y -17.308,Z -34.920,A -90.000,B 90.000,C 0.000} C_DIS
LIN {X 107.311,Y -17.308,Z -34.835,A -90.000,B 90.000,C 0.000} C_DIS
LIN {X 107.359,Y -17.308,Z -34.755,A -90.000,B 90.000,C 0.000} C_DIS
LIN {X 107.400,Y -17.308,Z -34.678,A -90.000,B 90.000,C 0.000} C_DIS
LIN {X 107.449,Y -17.308,Z -34.572,A -90.000,B 90.000,C 0.000} C_DIS
LIN {X 107.473,Y -17.308,Z -34.506,A -90.000,B 90.000,C 0.000} C_DIS
LIN {X 107.509,Y -17.308,Z -34.388,A -90.000,B 90.000,C 0.000} C_DIS
LIN {X 107.531,Y -17.308,Z -34.287,A -90.000,B 90.000,C 0.000} C_DIS
LIN {X 107.551,Y -17.308,Z -34.167,A -90.000,B 90.000,C 0.000} C_DIS
LIN {X 107.565,Y -17.308,Z -34.109,A -90.000,B 90.000,C 0.000} C_DIS
LIN {X 107.581,Y -17.308,Z -34.076,A -90.000,B 90.000,C 0.000} C_DIS
LIN {X 107.594,Y -17.308,Z -34.060,A -90.000,B 90.000,C 0.000} C_DIS
LIN {X 107.612,Y -17.308,Z -34.048,A -90.000,B 90.000,C 0.000} C_DIS
LIN {X 107.634,Y -17.308,Z -34.040,A -90.000,B 90.000,C 0.000} C_DIS
LIN {X 107.678,Y -17.308,Z -34.036,A -90.000,B 90.000,C 0.000} C_DIS
LIN {X 107.714,Y -17.308,Z -34.039,A -90.000,B 90.000,C 0.000} C_DIS
LIN {X 107.759,Y -17.308,Z -34.047,A -90.000,B 90.000,C 0.000} C_DIS
LIN {X 107.872,Y -17.308,Z -34.074,A -90.000,B 90.000,C 0.000} C_DIS
LIN {X 108.023,Y -17.308,Z -34.118,A -90.000,B 90.000,C 0.000} C_DIS
LIN {X 109.132,Y -17.308,Z -34.467,A -90.000,B 90.000,C 0.000} C_DIS
LIN {X 109.565,Y -17.308,Z -34.597,A -90.000,B 90.000,C 0.000} C_DIS
LIN {X 110.074,Y -17.308,Z -34.744,A -90.000,B 90.000,C 0.000} C_DIS
LIN {X 110.990,Y -17.308,Z -34.997,A -90.000,B 90.000,C 0.000} C_DIS
LIN {X 112.110,Y -17.308,Z -35.288,A -90.000,B 90.000,C 0.000} C_DIS
LIN {X 112.241,Y -17.308,Z -35.321,A -90.000,B 90.000,C 0.000} C_DIS
LIN {X 112.241,Y -60.000,Z -35.321,A -90.000,B 90.000,C 0.000} C_DIS
LIN {X 117.092,Y -60.000,Z -46.302,A -90.000,B 90.000,C 0.000} C_DIS
LIN {X 117.092,Y -17.308,Z -46.302,A -90.000,B 90.000,C 0.000} C_DIS
LIN {X 117.031,Y -17.308,Z -46.505,A -90.000,B 90.000,C 0.000} C_DIS
LIN {X 116.930,Y -17.306,Z -46.879,A -90.000,B 90.000,C 0.000} C_DIS
LIN {X 116.822,Y -17.308,Z -47.200,A -90.000,B 90.000,C 0.000} C_DIS
LIN {X 116.669,Y -17.308,Z -47.725,A -90.000,B 90.000,C 0.000} C_DIS
LIN {X 116.564,Y -17.308,Z -48.103,A -90.000,B 90.000,C 0.000} C_DIS
LIN {X 116.428,Y -17.308,Z -48.624,A -90.000,B 90.000,C 0.000} C_DIS
LIN {X 116.424,Y -17.308,Z -48.628,A -90.000,B 90.000,C 0.000} C_DIS
LIN {X 116.402,Y -17.308,Z -48.626,A -90.000,B 90.000,C 0.000} C_DIS
LIN {X 116.379,Y -17.308,Z -48.638,A -90.000,B 90.000,C 0.000} C_DIS
LIN {X 116.341,Y -17.308,Z -48.671,A -90.000,B 90.000,C 0.000} C_DIS
LIN {X 116.307,Y -17.308,Z -48.711,A -90.000,B 90.000,C 0.000} C_DIS
LIN {X 116.210,Y -17.308,Z -48.843,A -90.000,B 90.000,C 0.000} C_DIS
LIN {X 116.068,Y -17.308,Z -49.069,A -90.000,B 90.000,C 0.000} C_DIS
LIN {X 115.872,Y -17.308,Z -49.410,A -90.000,B 90.000,C 0.000} C_DIS
LIN {X 115.751,Y -17.308,Z -49.632,A -90.000,B 90.000,C 0.000} C_DIS
LIN {X 115.456,Y -17.308,Z -50.192,A -90.000,B 90.000,C 0.000} C_DIS
LIN {X 115.280,Y -17.308,Z -50.537,A -90.000,B 90.000,C 0.000} C_DIS
LIN {X 115.199,Y -17.308,Z -50.697,A -90.000,B 90.000,C 0.000} C_DIS
LIN {X 115.199,Y -60.000,Z -50.697,A -90.000,B 90.000,C 0.000} C_DIS
LIN {X 110.671,Y -60.000,Z -62.597,A -90.000,B 90.000,C 0.000} C_DIS
LIN {X 110.671,Y -17.308,Z -62.597,A -90.000,B 90.000,C 0.000} C_DIS
LIN {X 110.455,Y -17.308,Z -63.363,A -90.000,B 90.000,C 0.000} C_DIS
LIN {X 110.455,Y -60.000,Z -63.363,A -90.000,B 90.000,C 0.000} C_DIS
LIN {X 99.843,Y -60.000,Z -87.123,A -90.000,B 90.000,C 0.000} C_DIS
LIN {X 99.843,Y -17.308,Z -87.123,A -90.000,B 90.000,C 0.000} C_DIS
LIN {X 99.858,Y -17.308,Z -87.310,A -90.000,B 90.000,C 0.000} C_DIS
LIN {X 99.858,Y -60.000,Z -87.310,A -90.000,B 90.000,C 0.000} C_DIS
LIN {X -3.690,Y -60.000,Z -36.816,A -90.000,B 90.000,C 0.000} C_DIS
LIN {X -3.690,Y -17.308,Z -36.816,A -90.000,B 90.000,C 0.000} C_DIS
LIN {X -3.084,Y -17.362,Z -36.962,A -90.000,B 90.000,C 0.000} C_DIS
LIN {X -2.710,Y -17.384,Z -37.035,A -90.000,B 90.000,C 0.000} C_DIS
LIN {X -2.307,Y -17.400,Z -37.105,A -90.000,B 90.000,C 0.000} C_DIS
LIN {X -2.108,Y -17.407,Z -37.139,A -90.000,B 90.000,C 0.000} C_DIS
LIN {X -1.070,Y -17.405,Z -37.260,A -90.000,B 90.000,C 0.000} C_DIS
LIN {X -1.000,Y -17.406,Z -37.268,A -90.000,B 90.000,C 0.000} C_DIS
LIN {X 0.548,Y -17.378,Z -37.357,A -90.000,B 90.000,C 0.000} C_DIS
LIN {X 1.093,Y -17.370,Z -37.392,A -90.000,B 90.000,C 0.000} C_DIS
LIN {X 2.515,Y -17.313,Z -37.455,A -90.000,B 90.000,C 0.000} C_DIS
LIN {X 2.590,Y -17.308,Z -37.459,A -90.000,B 90.000,C 0.000} C_DIS
LIN {X 2.590,Y -60.000,Z -37.459,A -90.000,B 90.000,C 0.000} C_DIS
LIN {X -62.083,Y -60.000,Z -26.174,A -90.000,B 90.000,C 0.000} C_DIS
LIN {X -62.083,Y -17.308,Z -26.174,A -90.000,B 90.000,C 0.000} C_DIS
LIN {X -62.057,Y -17.320,Z -26.223,A -90.000,B 90.000,C 0.000} C_DIS
LIN {X -61.982,Y -17.364,Z -26.367,A -90.000,B 90.000,C 0.000} C_DIS
LIN {X -61.936,Y -17.392,Z -26.457,A -90.000,B 90.000,C 0.000} C_DIS
LIN {X -61.836,Y -17.459,Z -26.665,A -90.000,B 90.000,C 0.000} C_DIS
LIN {X -61.705,Y -17.521,Z -26.886,A -90.000,B 90.000,C 0.000} C_DIS
LIN {X -61.654,Y -17.545,Z -26.975,A -90.000,B 90.000,C 0.000} C_DIS
LIN {X -61.524,Y -17.547,Z -27.066,A -90.000,B 90.000,C 0.000} C_DIS
LIN {X -61.349,Y -17.565,Z -27.177,A -90.000,B 90.000,C 0.000} C_DIS
LIN {X -60.525,Y -17.576,Z -27.557,A -90.000,B 90.000,C 0.000} C_DIS
LIN {X -60.349,Y -17.587,Z -27.634,A -90.000,B 90.000,C 0.000} C_DIS
LIN {X -58.969,Y -17.614,Z -28.120,A -90.000,B 90.000,C 0.000} C_DIS
LIN {X -58.840,Y -17.618,Z -28.162,A -90.000,B 90.000,C 0.000} C_DIS
LIN {X -58.476,Y -17.621,Z -28.267,A -90.000,B 90.000,C 0.000} C_DIS
LIN {X -57.352,Y -17.635,Z -28.602,A -90.000,B 90.000,C 0.000} C_DIS
LIN {X -57.008,Y -17.643,Z -28.709,A -90.000,B 90.000,C 0.000} C_DIS
LIN {X -56.728,Y -17.655,Z -28.795,A -90.000,B 90.000,C 0.000} C_DIS
LIN {X -55.564,Y -17.670,Z -29.078,A -90.000,B 90.000,C 0.000} C_DIS
LIN {X -54.958,Y -17.675,Z -29.221,A -90.000,B 90.000,C 0.000} C_DIS
LIN {X -54.838,Y -17.677,Z -29.249,A -90.000,B 90.000,C 0.000} C_DIS
LIN {X -54.527,Y -17.672,Z -29.298,A -90.000,B 90.000,C 0.000} C_DIS
LIN {X -53.273,Y -17.630,Z -29.508,A -90.000,B 90.000,C 0.000} C_DIS
LIN {X -52.532,Y -17.618,Z -29.625,A -90.000,B 90.000,C 0.000} C_DIS
LIN {X -51.860,Y -17.576,Z -29.676,A -90.000,B 90.000,C 0.000} C_DIS
LIN {X -51.439,Y -17.563,Z -29.701,A -90.000,B 90.000,C 0.000} C_DIS
LIN {X -51.040,Y -17.535,Z -29.734,A -90.000,B 90.000,C 0.000} C_DIS
LIN {X -50.634,Y -17.511,Z -29.775,A -90.000,B 90.000,C 0.000} C_DIS
LIN {X -50.354,Y -17.496,Z -29.805,A -90.000,B 90.000,C 0.000} C_DIS
LIN {X -49.670,Y -17.474,Z -29.868,A -90.000,B 90.000,C 0.000} C_DIS
LIN {X -49.473,Y -17.451,Z -29.858,A -90.000,B 90.000,C 0.000} C_DIS
LIN {X -49.179,Y -17.423,Z -29.855,A -90.000,B 90.000,C 0.000} C_DIS
LIN {X -48.354,Y -17.378,Z -29.871,A -90.000,B 90.000,C 0.000} C_DIS
LIN {X -48.091,Y -17.367,Z -29.884,A -90.000,B 90.000,C 0.000} C_DIS
LIN {X -46.632,Y -17.331,Z -29.999,A -90.000,B 90.000,C 0.000} C_DIS
LIN {X -46.217,Y -17.308,Z -30.012,A -90.000,B 90.000,C 0.000} C_DIS
LIN {X -46.217,Y -60.000,Z -30.012,A -90.000,B 90.000,C 0.000} C_DIS
LIN {X -112.144,Y -60.000,Z -243.561,A -90.000,B 90.000,C 0.000} C_DIS
LIN {X -112.144,Y -17.674,Z -243.561,A -90.000,B 90.000,C 0.000} C_DIS
LIN {X -112.115,Y -17.615,Z -243.444,A -90.000,B 90.000,C 0.000} C_DIS
LIN {X -112.062,Y -17.528,Z -243.263,A -90.000,B 90.000,C 0.000} C_DIS
LIN {X -112.014,Y -17.464,Z -243.124,A -90.000,B 90.000,C 0.000} C_DIS
LIN {X -111.955,Y -17.396,Z -242.970,A -90.000,B 90.000,C 0.000} C_DIS
LIN {X -111.898,Y -17.340,Z -242.838,A -90.000,B 90.000,C 0.000} C_DIS
LIN {X -111.862,Y -17.308,Z -242.760,A -90.000,B 90.000,C 0.000} C_DIS
LIN {X -111.843,Y -17.288,Z -242.705,A -90.000,B 90.000,C 0.000} C_DIS
LIN {X -111.809,Y -17.249,Z -242.618,A -90.000,B 90.000,C 0.000} C_DIS
LIN {X -111.794,Y -17.215,Z -242.551,A -90.000,B 90.000,C 0.000} C_DIS
LIN {X -111.794,Y -17.192,Z -242.514,A -90.000,B 90.000,C 0.000} C_DIS
LIN {X -111.803,Y -17.173,Z -242.487,A -90.000,B 90.000,C 0.000} C_DIS
LIN {X -111.820,Y -17.155,Z -242.469,A -90.000,B 90.000,C 0.000} C_DIS
LIN {X -111.845,Y -17.138,Z -242.460,A -90.000,B 90.000,C 0.000} C_DIS
LIN {X -111.865,Y -17.130,Z -242.460,A -90.000,B 90.000,C 0.000} C_DIS
LIN {X -111.888,Y -17.122,Z -242.463,A -90.000,B 90.000,C 0.000} C_DIS
LIN {X -111.941,Y -17.110,Z -242.480,A -90.000,B 90.000,C 0.000} C_DIS
LIN {X -112.005,Y -17.101,Z -242.511,A -90.000,B 90.000,C 0.000} C_DIS
LIN {X -112.077,Y -17.096,Z -242.553,A -90.000,B 90.000,C 0.000} C_DIS
LIN {X -112.198,Y -17.094,Z -242.635,A -90.000,B 90.000,C 0.000} C_DIS
LIN {X -112.285,Y -17.096,Z -242.701,A -90.000,B 90.000,C 0.000} C_DIS
LIN {X -112.469,Y -17.108,Z -242.849,A -90.000,B 90.000,C 0.000} C_DIS
LIN {X -112.563,Y -17.117,Z -242.930,A -90.000,B 90.000,C 0.000} C_DIS
LIN {X -112.749,Y -17.140,Z -243.098,A -90.000,B 90.000,C 0.000} C_DIS
LIN {X -112.837,Y -17.153,Z -243.183,A -90.000,B 90.000,C 0.000} C_DIS
LIN {X -113.000,Y -17.182,Z -243.345,A -90.000,B 90.000,C 0.000} C_DIS
LIN {X -113.135,Y -17.212,Z -243.490,A -90.000,B 90.000,C 0.000} C_DIS
LIN {X -113.188,Y -17.227,Z -243.552,A -90.000,B 90.000,C 0.000} C_DIS
LIN {X -113.246,Y -17.249,Z -243.628,A -90.000,B 90.000,C 0.000} C_DIS
LIN {X -113.269,Y -17.262,Z -243.666,A -90.000,B 90.000,C 0.000} C_DIS
LIN {X -113.274,Y -17.268,Z -243.680,A -90.000,B 90.000,C 0.000} C_DIS
LIN {X -113.276,Y -17.274,Z -243.692,A -90.000,B 90.000,C 0.000} C_DIS
LIN {X -113.274,Y -17.280,Z -243.700,A -90.000,B 90.000,C 0.000} C_DIS
LIN {X -113.268,Y -17.285,Z -243.704,A -90.000,B 90.000,C 0.000} C_DIS
LIN {X -113.258,Y -17.290,Z -243.705,A -90.000,B 90.000,C 0.000} C_DIS
LIN {X -113.224,Y -17.298,Z -243.695,A -90.000,B 90.000,C 0.000} C_DIS
LIN {X -113.172,Y -17.304,Z -243.668,A -90.000,B 90.000,C 0.000} C_DIS
LIN {X -113.099,Y -17.308,Z -243.623,A -90.000,B 90.000,C 0.000} C_DIS
LIN {X -113.002,Y -17.308,Z -243.561,A -90.000,B 90.000,C 0.000} C_DIS
LIN {X -110.034,Y -17.308,Z -241.472,A -90.000,B 90.000,C 0.000} C_DIS
LIN {X -106.317,Y -17.308,Z -238.832,A -90.000,B 90.000,C 0.000} C_DIS
LIN {X -98.759,Y -17.308,Z -233.504,A -90.000,B 90.000,C 0.000} C_DIS
LIN {X -98.129,Y -17.308,Z -233.065,A -90.000,B 90.000,C 0.000} C_DIS
LIN {X -95.634,Y -17.308,Z -231.332,A -90.000,B 90.000,C 0.000} C_DIS
LIN {X -91.495,Y -17.308,Z -228.490,A -90.000,B 90.000,C 0.000} C_DIS
LIN {X -90.620,Y -17.308,Z -227.894,A -90.000,B 90.000,C 0.000} C_DIS
LIN {X -83.819,Y -17.308,Z -223.319,A -90.000,B 90.000,C 0.000} C_DIS
LIN {X -82.506,Y -17.308,Z -222.441,A -90.000,B 90.000,C 0.000} C_DIS
LIN {X -74.304,Y -17.308,Z -217.061,A -90.000,B 90.000,C 0.000} C_DIS
LIN {X -69.942,Y -17.308,Z -214.219,A -90.000,B 90.000,C 0.000} C_DIS
LIN {X -66.292,Y -17.308,Z -211.846,A -90.000,B 90.000,C 0.000} C_DIS
LIN {X -58.845,Y -17.308,Z -206.963,A -90.000,B 90.000,C 0.000} C_DIS
LIN {X -56.314,Y -17.308,Z -205.267,A -90.000,B 90.000,C 0.000} C_DIS
LIN {X -52.133,Y -17.308,Z -202.523,A -90.000,B 90.000,C 0.000} C_DIS
LIN {X -50.014,Y -17.308,Z -201.066,A -90.000,B 90.000,C 0.000} C_DIS
LIN {X -46.615,Y -17.308,Z -198.767,A -90.000,B 90.000,C 0.000} C_DIS
LIN {X -46.159,Y -17.308,Z -198.450,A -90.000,B 90.000,C 0.000} C_DIS
LIN {X -42.255,Y -17.308,Z -195.686,A -90.000,B 90.000,C 0.000} C_DIS
LIN {X -41.519,Y -17.308,Z -195.153,A -90.000,B 90.000,C 0.000} C_DIS
LIN {X -38.462,Y -17.308,Z -192.893,A -90.000,B 90.000,C 0.000} C_DIS
LIN {X -37.890,Y -17.308,Z -192.466,A -90.000,B 90.000,C 0.000} C_DIS
LIN {X -35.083,Y -17.308,Z -190.320,A -90.000,B 90.000,C 0.000} C_DIS
LIN {X -32.740,Y -17.308,Z -188.500,A -90.000,B 90.000,C 0.000} C_DIS
LIN {X -31.933,Y -17.308,Z -187.887,A -90.000,B 90.000,C 0.000} C_DIS
LIN {X -29.756,Y -17.308,Z -186.140,A -90.000,B 90.000,C 0.000} C_DIS
LIN {X -29.007,Y -17.308,Z -185.551,A -90.000,B 90.000,C 0.000} C_DIS
LIN {X -26.924,Y -17.308,Z -183.792,A -90.000,B 90.000,C 0.000} C_DIS
LIN {X -26.272,Y -17.308,Z -183.252,A -90.000,B 90.000,C 0.000} C_DIS
LIN {X -24.261,Y -17.308,Z -181.434,A -90.000,B 90.000,C 0.000} C_DIS
LIN {X -23.821,Y -17.308,Z -181.044,A -90.000,B 90.000,C 0.000} C_DIS
LIN {X -23.503,Y -17.308,Z -180.737,A -90.000,B 90.000,C 0.000} C_DIS
LIN {X -21.567,Y -17.308,Z -178.839,A -90.000,B 90.000,C 0.000} C_DIS
LIN {X -21.087,Y -17.308,Z -178.328,A -90.000,B 90.000,C 0.000} C_DIS
LIN {X -19.295,Y -17.308,Z -176.398,A -90.000,B 90.000,C 0.000} C_DIS
LIN {X -19.105,Y -17.308,Z -176.173,A -90.000,B 90.000,C 0.000} C_DIS
LIN {X -17.426,Y -17.308,Z -174.154,A -90.000,B 90.000,C 0.000} C_DIS
LIN {X -17.063,Y -17.308,Z -173.666,A -90.000,B 90.000,C 0.000} C_DIS
LIN {X -15.596,Y -17.308,Z -171.656,A -90.000,B 90.000,C 0.000} C_DIS
LIN {X -14.129,Y -17.308,Z -169.312,A -90.000,B 90.000,C 0.000} C_DIS
LIN {X -13.984,Y -17.308,Z -169.085,A -90.000,B 90.000,C 0.000} C_DIS
LIN {X -13.041,Y -17.308,Z -167.258,A -90.000,B 90.000,C 0.000} C_DIS
LIN {X -12.735,Y -17.308,Z -166.670,A -90.000,B 90.000,C 0.000} C_DIS
LIN {X -11.894,Y -17.308,Z -164.530,A -90.000,B 90.000,C 0.000} C_DIS
LIN {X -11.542,Y -17.308,Z -162.923,A -90.000,B 90.000,C 0.000} C_DIS
LIN {X -11.546,Y -17.308,Z -162.811,A -90.000,B 90.000,C 0.000} C_DIS
LIN {X -11.581,Y -17.308,Z -161.904,A -90.000,B 90.000,C 0.000} C_DIS
LIN {X -11.784,Y -17.308,Z -161.278,A -90.000,B 90.000,C 0.000} C_DIS
LIN {X -11.996,Y -17.308,Z -160.929,A -90.000,B 90.000,C 0.000} C_DIS
LIN {X -12.231,Y -17.308,Z -160.538,A -90.000,B 90.000,C 0.000} C_DIS
LIN {X -12.622,Y -17.308,Z -160.060,A -90.000,B 90.000,C 0.000} C_DIS
LIN {X -12.896,Y -17.308,Z -159.696,A -90.000,B 90.000,C 0.000} C_DIS
LIN {X -13.011,Y -17.308,Z -159.530,A -90.000,B 90.000,C 0.000} C_DIS
LIN {X -13.623,Y -17.308,Z -158.835,A -90.000,B 90.000,C 0.000} C_DIS
LIN {X -13.817,Y -17.308,Z -158.584,A -90.000,B 90.000,C 0.000} C_DIS
LIN {X -13.967,Y -17.308,Z -158.387,A -90.000,B 90.000,C 0.000} C_DIS
LIN {X -14.722,Y -17.308,Z -157.599,A -90.000,B 90.000,C 0.000} C_DIS
LIN {X -15.105,Y -17.308,Z -157.140,A -90.000,B 90.000,C 0.000} C_DIS
LIN {X -15.783,Y -17.308,Z -156.485,A -90.000,B 90.000,C 0.000} C_DIS
LIN {X -16.217,Y -17.308,Z -156.038,A -90.000,B 90.000,C 0.000} C_DIS
LIN {X -16.634,Y -17.308,Z -155.594,A -90.000,B 90.000,C 0.000} C_DIS
LIN {X -17.836,Y -17.308,Z -154.496,A -90.000,B 90.000,C 0.000} C_DIS
LIN {X -18.633,Y -17.308,Z -153.715,A -90.000,B 90.000,C 0.000} C_DIS
LIN {X -20.347,Y -17.308,Z -152.209,A -90.000,B 90.000,C 0.000} C_DIS
LIN {X -23.381,Y -17.308,Z -149.425,A -90.000,B 90.000,C 0.000} C_DIS
LIN {X -24.683,Y -17.308,Z -148.192,A -90.000,B 90.000,C 0.000} C_DIS
LIN {X -25.023,Y -17.308,Z -147.859,A -90.000,B 90.000,C 0.000} C_DIS
LIN {X -27.043,Y -17.308,Z -145.804,A -90.000,B 90.000,C 0.000} C_DIS
LIN {X -28.147,Y -17.308,Z -144.658,A -90.000,B 90.000,C 0.000} C_DIS
LIN {X -28.300,Y -17.308,Z -144.497,A -90.000,B 90.000,C 0.000} C_DIS
LIN {X -28.474,Y -17.308,Z -144.302,A -90.000,B 90.000,C 0.000} C_DIS
LIN {X -31.151,Y -17.308,Z -141.085,A -90.000,B 90.000,C 0.000} C_DIS
LIN {X -31.526,Y -17.308,Z -140.627,A -90.000,B 90.000,C 0.000} C_DIS
LIN {X -31.814,Y -17.308,Z -140.239,A -90.000,B 90.000,C 0.000} C_DIS
LIN {X -32.079,Y -17.308,Z -139.820,A -90.000,B 90.000,C 0.000} C_DIS
LIN {X -33.808,Y -17.308,Z -137.128,A -90.000,B 90.000,C 0.000} C_DIS
LIN {X -34.357,Y -17.308,Z -136.267,A -90.000,B 90.000,C 0.000} C_DIS
LIN {X -34.561,Y -17.308,Z -135.922,A -90.000,B 90.000,C 0.000} C_DIS
LIN {X -36.383,Y -17.308,Z -132.377,A -90.000,B 90.000,C 0.000} C_DIS
LIN {X -36.712,Y -17.308,Z -131.733,A -90.000,B 90.000,C 0.000} C_DIS
LIN {X -38.323,Y -17.308,Z -128.030,A -90.000,B 90.000,C 0.000} C_DIS
LIN {X -39.494,Y -17.308,Z -125.139,A -90.000,B 90.000,C 0.000} C_DIS
LIN {X -39.782,Y -17.308,Z -124.415,A -90.000,B 90.000,C 0.000} C_DIS
LIN {X -40.067,Y -17.308,Z -123.749,A -90.000,B 90.000,C 0.000} C_DIS
LIN {X -40.570,Y -17.308,Z -122.555,A -90.000,B 90.000,C 0.000} C_DIS
LIN {X -41.093,Y -17.308,Z -121.474,A -90.000,B 90.000,C 0.000} C_DIS
LIN {X -41.384,Y -17.308,Z -120.923,A -90.000,B 90.000,C 0.000} C_DIS
LIN {X -41.673,Y -17.308,Z -120.444,A -90.000,B 90.000,C 0.000} C_DIS
LIN {X -42.214,Y -17.308,Z -119.604,A -90.000,B 90.000,C 0.000} C_DIS
LIN {X -42.545,Y -17.308,Z -119.147,A -90.000,B 90.000,C 0.000} C_DIS
LIN {X -43.309,Y -17.308,Z -118.127,A -90.000,B 90.000,C 0.000} C_DIS
LIN {X -45.159,Y -17.308,Z -115.835,A -90.000,B 90.000,C 0.000} C_DIS
LIN {X -47.502,Y -17.308,Z -112.961,A -90.000,B 90.000,C 0.000} C_DIS
LIN {X -48.730,Y -17.308,Z -111.422,A -90.000,B 90.000,C 0.000} C_DIS
LIN {X -50.008,Y -17.308,Z -109.832,A -90.000,B 90.000,C 0.000} C_DIS
LIN {X -52.039,Y -17.308,Z -107.203,A -90.000,B 90.000,C 0.000} C_DIS
LIN {X -52.598,Y -17.308,Z -106.475,A -90.000,B 90.000,C 0.000} C_DIS
LIN {X -52.812,Y -17.308,Z -106.187,A -90.000,B 90.000,C 0.000} C_DIS
LIN {X -54.743,Y -17.308,Z -103.543,A -90.000,B 90.000,C 0.000} C_DIS
LIN {X -55.389,Y -17.308,Z -102.668,A -90.000,B 90.000,C 0.000} C_DIS
LIN {X -56.006,Y -17.308,Z -101.806,A -90.000,B 90.000,C 0.000} C_DIS
LIN {X -57.155,Y -17.308,Z -100.230,A -90.000,B 90.000,C 0.000} C_DIS
LIN {X -57.520,Y -17.308,Z -99.727,A -90.000,B 90.000,C 0.000} C_DIS
LIN {X -57.826,Y -17.308,Z -99.314,A -90.000,B 90.000,C 0.000} C_DIS
LIN {X -58.959,Y -17.308,Z -97.770,A -90.000,B 90.000,C 0.000} C_DIS
LIN {X -59.869,Y -17.308,Z -96.559,A -90.000,B 90.000,C 0.000} C_DIS
LIN {X -60.343,Y -17.308,Z -95.935,A -90.000,B 90.000,C 0.000} C_DIS
LIN {X -61.349,Y -17.308,Z -94.629,A -90.000,B 90.000,C 0.000} C_DIS
LIN {X -61.823,Y -17.308,Z -94.009,A -90.000,B 90.000,C 0.000} C_DIS
LIN {X -62.040,Y -17.308,Z -93.730,A -90.000,B 90.000,C 0.000} C_DIS
LIN {X -63.280,Y -17.308,Z -92.193,A -90.000,B 90.000,C 0.000} C_DIS
LIN {X -64.004,Y -17.308,Z -91.301,A -90.000,B 90.000,C 0.000} C_DIS
LIN {X -64.673,Y -17.308,Z -90.531,A -90.000,B 90.000,C 0.000} C_DIS
LIN {X -65.734,Y -17.308,Z -89.295,A -90.000,B 90.000,C 0.000} C_DIS
LIN {X -66.252,Y -17.308,Z -88.737,A -90.000,B 90.000,C 0.000} C_DIS
LIN {X -67.322,Y -17.308,Z -87.574,A -90.000,B 90.000,C 0.000} C_DIS
LIN {X -67.634,Y -17.308,Z -87.277,A -90.000,B 90.000,C 0.000} C_DIS
LIN {X -67.974,Y -17.308,Z -86.944,A -90.000,B 90.000,C 0.000} C_DIS
LIN {X -69.009,Y -17.308,Z -85.897,A -90.000,B 90.000,C 0.000} C_DIS
LIN {X -69.660,Y -17.308,Z -85.292,A -90.000,B 90.000,C 0.000} C_DIS
LIN {X -70.514,Y -17.308,Z -84.493,A -90.000,B 90.000,C 0.000} C_DIS
LIN {X -70.873,Y -17.308,Z -84.175,A -90.000,B 90.000,C 0.000} C_DIS
LIN {X -72.155,Y -17.308,Z -83.066,A -90.000,B 90.000,C 0.000} C_DIS
LIN {X -72.488,Y -17.308,Z -82.793,A -90.000,B 90.000,C 0.000} C_DIS
LIN {X -73.653,Y -17.308,Z -81.884,A -90.000,B 90.000,C 0.000} C_DIS
LIN {X -74.304,Y -17.308,Z -81.407,A -90.000,B 90.000,C 0.000} C_DIS
LIN {X -74.712,Y -17.308,Z -81.142,A -90.000,B 90.000,C 0.000} C_DIS
LIN {X -75.946,Y -17.308,Z -80.373,A -90.000,B 90.000,C 0.000} C_DIS
LIN {X -76.928,Y -17.308,Z -79.896,A -90.000,B 90.000,C 0.000} C_DIS
LIN {X -77.441,Y -17.308,Z -79.656,A -90.000,B 90.000,C 0.000} C_DIS
LIN {X -78.053,Y -17.308,Z -79.404,A -90.000,B 90.000,C 0.000} C_DIS
LIN {X -79.064,Y -17.308,Z -78.967,A -90.000,B 90.000,C 0.000} C_DIS
LIN {X -79.135,Y -17.308,Z -78.939,A -90.000,B 90.000,C 0.000} C_DIS
LIN {X -79.376,Y -17.308,Z -78.839,A -90.000,B 90.000,C 0.000} C_DIS
LIN {X -80.913,Y -17.308,Z -78.146,A -90.000,B 90.000,C 0.000} C_DIS
LIN {X -81.327,Y -17.308,Z -77.927,A -90.000,B 90.000,C 0.000} C_DIS
LIN {X -81.912,Y -17.308,Z -77.605,A -90.000,B 90.000,C 0.000} C_DIS
LIN {X -82.891,Y -17.308,Z -77.098,A -90.000,B 90.000,C 0.000} C_DIS
LIN {X -83.530,Y -17.308,Z -76.701,A -90.000,B 90.000,C 0.000} C_DIS
LIN {X -83.932,Y -17.308,Z -76.445,A -90.000,B 90.000,C 0.000} C_DIS
LIN {X -84.695,Y -17.308,Z -75.904,A -90.000,B 90.000,C 0.000} C_DIS
LIN {X -85.269,Y -17.308,Z -75.493,A -90.000,B 90.000,C 0.000} C_DIS
LIN {X -85.516,Y -17.308,Z -75.298,A -90.000,B 90.000,C 0.000} C_DIS
LIN {X -86.129,Y -17.308,Z -74.835,A -90.000,B 90.000,C 0.000} C_DIS
LIN {X -86.696,Y -17.308,Z -74.401,A -90.000,B 90.000,C 0.000} C_DIS
LIN {X -87.032,Y -17.308,Z -74.132,A -90.000,B 90.000,C 0.000} C_DIS
LIN {X -87.538,Y -17.308,Z -73.755,A -90.000,B 90.000,C 0.000} C_DIS
LIN {X -87.693,Y -17.308,Z -73.629,A -90.000,B 90.000,C 0.000} C_DIS
LIN {X -88.346,Y -17.308,Z -73.114,A -90.000,B 90.000,C 0.000} C_DIS
LIN {X -89.013,Y -17.308,Z -72.553,A -90.000,B 90.000,C 0.000} C_DIS
LIN {X -89.689,Y -17.308,Z -71.978,A -90.000,B 90.000,C 0.000} C_DIS
LIN {X -89.732,Y -17.308,Z -71.946,A -90.000,B 90.000,C 0.000} C_DIS
LIN {X -90.064,Y -17.308,Z -71.682,A -90.000,B 90.000,C 0.000} C_DIS
LIN {X -90.368,Y -17.308,Z -71.430,A -90.000,B 90.000,C 0.000} C_DIS
LIN {X -90.480,Y -17.308,Z -71.353,A -90.000,B 90.000,C 0.000} C_DIS
LIN {X -90.811,Y -17.308,Z -71.114,A -90.000,B 90.000,C 0.000} C_DIS
LIN {X -90.889,Y -17.308,Z -71.056,A -90.000,B 90.000,C 0.000} C_DIS
LIN {X -91.301,Y -17.308,Z -70.809,A -90.000,B 90.000,C 0.000} C_DIS
LIN {X -91.562,Y -17.308,Z -70.670,A -90.000,B 90.000,C 0.000} C_DIS
LIN {X -91.974,Y -17.308,Z -70.445,A -90.000,B 90.000,C 0.000} C_DIS
LIN {X -92.158,Y -17.308,Z -70.357,A -90.000,B 90.000,C 0.000} C_DIS
LIN {X -92.809,Y -17.308,Z -70.033,A -90.000,B 90.000,C 0.000} C_DIS
LIN {X -92.943,Y -17.308,Z -69.960,A -90.000,B 90.000,C 0.000} C_DIS
LIN {X -93.548,Y -17.308,Z -69.663,A -90.000,B 90.000,C 0.000} C_DIS
LIN {X -93.764,Y -17.308,Z -69.545,A -90.000,B 90.000,C 0.000} C_DIS
LIN {X -93.832,Y -17.308,Z -69.510,A -90.000,B 90.000,C 0.000} C_DIS
LIN {X -94.038,Y -17.308,Z -69.393,A -90.000,B 90.000,C 0.000} C_DIS
LIN {X -94.514,Y -17.308,Z -69.183,A -90.000,B 90.000,C 0.000} C_DIS
LIN {X -94.636,Y -17.308,Z -69.113,A -90.000,B 90.000,C 0.000} C_DIS
LIN {X -94.914,Y -17.308,Z -68.977,A -90.000,B 90.000,C 0.000} C_DIS
LIN {X -95.072,Y -17.308,Z -68.924,A -90.000,B 90.000,C 0.000} C_DIS
LIN {X -95.290,Y -17.308,Z -68.824,A -90.000,B 90.000,C 0.000} C_DIS
LIN {X -96.023,Y -17.308,Z -68.545,A -90.000,B 90.000,C 0.000} C_DIS
LIN {X -96.423,Y -17.308,Z -68.367,A -90.000,B 90.000,C 0.000} C_DIS
LIN {X -96.602,Y -17.308,Z -68.322,A -90.000,B 90.000,C 0.000} C_DIS
LIN {X -96.933,Y -17.308,Z -68.217,A -90.000,B 90.000,C 0.000} C_DIS
LIN {X -97.882,Y -17.308,Z -67.875,A -90.000,B 90.000,C 0.000} C_DIS
LIN {X -98.002,Y -17.308,Z -67.828,A -90.000,B 90.000,C 0.000} C_DIS
LIN {X -98.289,Y -17.308,Z -67.697,A -90.000,B 90.000,C 0.000} C_DIS
LIN {X -98.815,Y -17.308,Z -67.439,A -90.000,B 90.000,C 0.000} C_DIS
LIN {X -99.443,Y -17.308,Z -67.123,A -90.000,B 90.000,C 0.000} C_DIS
LIN {X -99.548,Y -17.308,Z -67.063,A -90.000,B 90.000,C 0.000} C_DIS
LIN {X -99.840,Y -17.308,Z -66.880,A -90.000,B 90.000,C 0.000} C_DIS
LIN {X -100.897,Y -17.308,Z -66.167,A -90.000,B 90.000,C 0.000} C_DIS
LIN {X -101.282,Y -17.308,Z -65.850,A -90.000,B 90.000,C 0.000} C_DIS
LIN {X -101.699,Y -17.308,Z -65.468,A -90.000,B 90.000,C 0.000} C_DIS
LIN {X -102.249,Y -17.308,Z -64.947,A -90.000,B 90.000,C 0.000} C_DIS
LIN {X -102.319,Y -17.308,Z -64.875,A -90.000,B 90.000,C 0.000} C_DIS
LIN {X -102.503,Y -17.308,Z -64.676,A -90.000,B 90.000,C 0.000} C_DIS
LIN {X -102.599,Y -17.308,Z -64.548,A -90.000,B 90.000,C 0.000} C_DIS
LIN {X -103.181,Y -17.308,Z -63.745,A -90.000,B 90.000,C 0.000} C_DIS
LIN {X -103.400,Y -17.308,Z -63.435,A -90.000,B 90.000,C 0.000} C_DIS
LIN {X -103.931,Y -17.308,Z -62.654,A -90.000,B 90.000,C 0.000} C_DIS
LIN {X -104.028,Y -17.308,Z -62.485,A -90.000,B 90.000,C 0.000} C_DIS
LIN {X -104.126,Y -17.308,Z -62.307,A -90.000,B 90.000,C 0.000} C_DIS
LIN {X -104.269,Y -17.308,Z -62.035,A -90.000,B 90.000,C 0.000} C_DIS
LIN {X -104.665,Y -17.308,Z -61.251,A -90.000,B 90.000,C 0.000} C_DIS
LIN {X -105.048,Y -17.308,Z -60.471,A -90.000,B 90.000,C 0.000} C_DIS
LIN {X -105.139,Y -17.308,Z -60.252,A -90.000,B 90.000,C 0.000} C_DIS
LIN {X -105.368,Y -17.308,Z -59.755,A -90.000,B 90.000,C 0.000} C_DIS
LIN {X -105.449,Y -17.308,Z -59.627,A -90.000,B 90.000,C 0.000} C_DIS
LIN {X -105.544,Y -17.308,Z -59.501,A -90.000,B 90.000,C 0.000} C_DIS
LIN {X -105.955,Y -17.308,Z -59.020,A -90.000,B 90.000,C 0.000} C_DIS
LIN {X -105.985,Y -17.308,Z -58.982,A -90.000,B 90.000,C 0.000} C_DIS
LIN {X -106.002,Y -17.308,Z -58.962,A -90.000,B 90.000,C 0.000} C_DIS
LIN {X -106.240,Y -17.308,Z -58.673,A -90.000,B 90.000,C 0.000} C_DIS
LIN {X -106.627,Y -17.308,Z -58.216,A -90.000,B 90.000,C 0.000} C_DIS
LIN {X -106.949,Y -17.308,Z -57.813,A -90.000,B 90.000,C 0.000} C_DIS
LIN {X -107.203,Y -17.308,Z -57.509,A -90.000,B 90.000,C 0.000} C_DIS
LIN {X -107.283,Y -17.308,Z -57.405,A -90.000,B 90.000,C 0.000} C_DIS
LIN {X -107.351,Y -17.308,Z -57.323,A -90.000,B 90.000,C 0.000} C_DIS
LIN {X -107.636,Y -17.308,Z -56.953,A -90.000,B 90.000,C 0.000} C_DIS
LIN {X -107.819,Y -17.308,Z -56.706,A -90.000,B 90.000,C 0.000} C_DIS
LIN {X -107.979,Y -17.308,Z -56.496,A -90.000,B 90.000,C 0.000} C_DIS
LIN {X -108.068,Y -17.308,Z -56.371,A -90.000,B 90.000,C 0.000} C_DIS
LIN {X -108.168,Y -17.308,Z -56.236,A -90.000,B 90.000,C 0.000} C_DIS
LIN {X -108.401,Y -17.308,Z -55.890,A -90.000,B 90.000,C 0.000} C_DIS
LIN {X -108.624,Y -17.308,Z -55.545,A -90.000,B 90.000,C 0.000} C_DIS
LIN {X -108.932,Y -17.308,Z -55.024,A -90.000,B 90.000,C 0.000} C_DIS
LIN {X -109.220,Y -17.308,Z -54.541,A -90.000,B 90.000,C 0.000} C_DIS
